C09148=1159.700,396.204,-85.224,-176.115,9.527,148.823
C09149=1159.704,395.957,-85.187,-176.115,9.525,148.822
C09150=1159.708,395.710,-85.150,-176.114,9.523,148.821
C09151=1159.712,395.462,-85.115,-176.114,9.520,148.821
C09152=1159.716,395.215,-85.078,-176.113,9.517,148.820
C09153=1159.720,394.968,-85.042,-176.112,9.515,148.819
C09154=1159.724,394.720,-85.005,-176.112,9.512,148.818
C09155=1159.728,394.473,-84.969,-176.112,9.510,148.818
C09156=1159.731,394.226,-84.932,-176.110,9.508,148.817
C09157=1159.736,393.979,-84.895,-176.110,9.505,148.816
C09158=1159.740,393.731,-84.859,-176.110,9.502,148.815
C09159=1159.743,393.484,-84.823,-176.109,9.500,148.814
C09160=1159.747,393.236,-84.786,-176.109,9.497,148.814
C09161=1159.750,392.989,-84.750,-176.108,9.495,148.813
C09162=1159.755,392.742,-84.713,-176.108,9.492,148.812
C09163=1159.759,392.495,-84.677,-176.107,9.489,148.811
C09164=1159.762,392.247,-84.641,-176.107,9.487,148.810
C09165=1159.766,392.000,-84.604,-176.107,9.484,148.809
C09166=1159.770,391.715,-84.562,-176.106,9.481,148.809
C09167=1159.775,391.429,-84.520,-176.106,9.477,148.808
C09168=1159.780,391.143,-84.479,-176.105,9.475,148.807
C09169=1159.784,390.858,-84.436,-176.106,9.471,148.806
C09170=1159.788,390.610,-84.400,-176.105,9.468,148.805
C09171=1159.792,390.363,-84.363,-176.105,9.465,148.804
C09172=1159.796,390.115,-84.326,-176.104,9.463,148.803
C09173=1159.799,389.867,-84.291,-176.104,9.460,148.803
C09174=1159.803,389.620,-84.254,-176.104,9.456,148.802
C09175=1159.807,389.373,-84.218,-176.104,9.454,148.801
C09176=1159.811,389.126,-84.181,-176.104,9.451,148.800
C09177=1159.814,388.879,-84.145,-176.104,9.448,148.799
C09178=1159.819,388.632,-84.108,-176.104,9.445,148.798
C09179=1159.822,388.384,-84.073,-176.104,9.441,148.798
C09180=1159.826,388.137,-84.036,-176.104,9.439,148.797
C09181=1159.831,387.889,-84.000,-176.104,9.435,148.796
C09182=1159.834,387.642,-83.964,-176.104,9.432,148.795
C09183=1159.838,387.395,-83.927,-176.104,9.429,148.794
C09184=1159.842,387.147,-83.891,-176.104,9.426,148.794
C09185=1159.846,386.900,-83.854,-176.104,9.423,148.793
C09186=1159.850,386.653,-83.819,-176.104,9.419,148.792
C09187=1159.854,386.406,-83.782,-176.105,9.416,148.791
C09188=1159.857,386.158,-83.746,-176.105,9.413,148.790
C09189=1159.861,385.911,-83.709,-176.105,9.410,148.790
C09190=1159.865,385.663,-83.674,-176.105,9.406,148.789
C09191=1159.869,385.416,-83.637,-176.106,9.403,148.788
C09192=1159.873,385.169,-83.601,-176.106,9.400,148.787
C09193=1159.877,384.921,-83.565,-176.106,9.396,148.786
C09194=1159.880,384.675,-83.528,-176.107,9.393,148.786
C09195=1159.885,384.427,-83.492,-176.107,9.389,148.785
C09196=1159.888,384.180,-83.456,-176.108,9.386,148.784
C09197=1159.892,383.932,-83.420,-176.109,9.382,148.783
C09198=1159.896,383.685,-83.384,-176.109,9.378,148.783
C09199=1159.900,383.437,-83.347,-176.110,9.375,148.782
C09200=1159.904,383.190,-83.312,-176.111,9.372,148.781
C09201=1159.908,382.943,-83.275,-176.112,9.368,148.780
C09202=1159.912,382.695,-83.239,-176.112,9.364,148.780
C09203=1159.916,382.448,-83.203,-176.112,9.361,148.779
C09204=1159.919,382.201,-83.167,-176.114,9.357,148.778
C09205=1159.923,381.954,-83.131,-176.114,9.354,148.777
C09206=1159.927,381.706,-83.095,-176.116,9.350,148.777
C09207=1159.931,381.458,-83.059,-176.116,9.346,148.776
C09208=1159.935,381.211,-83.022,-176.117,9.342,148.775
C09209=1159.939,380.964,-82.987,-176.118,9.339,148.775
C09210=1159.943,380.716,-82.950,-176.119,9.335,148.774
C09211=1159.947,380.470,-82.915,-176.120,9.332,148.773
C09212=1159.951,380.222,-82.879,-176.122,9.328,148.773
C09213=1159.955,379.975,-82.842,-176.123,9.324,148.772
C09214=1159.958,379.727,-82.807,-176.123,9.321,148.771
C09215=1159.963,379.480,-82.771,-176.125,9.317,148.771
C09216=1159.966,379.233,-82.734,-176.126,9.313,148.770
C09217=1159.970,378.985,-82.699,-176.127,9.309,148.769
C09218=1159.974,378.737,-82.663,-176.129,9.305,148.769
C09219=1159.978,378.490,-82.627,-176.130,9.302,148.768
C09220=1159.981,378.243,-82.591,-176.131,9.298,148.767
C09221=1159.986,377.995,-82.555,-176.133,9.294,148.767
C09222=1159.989,377.748,-82.519,-176.134,9.290,148.766
C09223=1159.994,377.501,-82.484,-176.135,9.286,148.765
C09224=1159.998,377.254,-82.447,-176.136,9.282,148.765
C09225=1160.001,377.006,-82.412,-176.138,9.278,148.764
C09226=1160.005,376.759,-82.376,-176.140,9.274,148.764
C09227=1160.009,376.511,-82.340,-176.141,9.270,148.763
C09228=1160.013,376.263,-82.304,-176.143,9.267,148.762
C09229=1160.016,376.017,-82.268,-176.144,9.263,148.762
C09230=1160.021,375.769,-82.232,-176.146,9.259,148.761
C09231=1160.025,375.522,-82.197,-176.147,9.255,148.761
C09232=1160.029,375.274,-82.161,-176.149,9.251,148.760
C09233=1160.032,375.027,-82.126,-176.150,9.247,148.759
C09234=1160.037,374.779,-82.089,-176.153,9.243,148.759
C09235=1160.040,374.532,-82.054,-176.154,9.239,148.758
C09236=1160.044,374.284,-82.018,-176.156,9.235,148.758
C09237=1160.048,374.037,-81.983,-176.158,9.232,148.757
C09238=1160.052,373.790,-81.948,-176.159,9.228,148.757
C09239=1160.056,373.542,-81.911,-176.161,9.223,148.756
C09240=1160.060,373.295,-81.876,-176.163,9.220,148.756
C09241=1160.064,373.047,-81.840,-176.165,9.216,148.755
C09242=1160.067,372.800,-81.805,-176.167,9.212,148.755
C09243=1160.072,372.553,-81.770,-176.169,9.208,148.754
C09244=1160.076,372.305,-81.734,-176.171,9.204,148.754
C09245=1160.080,372.057,-81.698,-176.172,9.200,148.753
C09246=1160.083,371.810,-81.662,-176.174,9.197,148.753
C09247=1160.087,371.562,-81.627,-176.177,9.192,148.752
C09248=1160.091,371.316,-81.592,-176.178,9.188,148.752
C09249=1160.095,371.068,-81.556,-176.180,9.185,148.751
C09250=1160.099,370.821,-81.521,-176.182,9.180,148.751
C09251=1160.102,370.573,-81.485,-176.184,9.177,148.750
C09252=1160.107,370.326,-81.449,-176.187,9.172,148.750
C09253=1160.111,370.079,-81.414,-176.189,9.169,148.750
C09254=1160.115,369.830,-81.379,-176.191,9.165,148.749
C09255=1160.119,369.583,-81.343,-176.193,9.161,148.749
C09256=1160.123,369.336,-81.308,-176.195,9.157,148.748
C09257=1160.126,369.089,-81.273,-176.197,9.153,148.748
C09258=1160.130,368.841,-81.237,-176.199,9.149,148.747
C09259=1160.134,368.593,-81.202,-176.202,9.145,148.747
C09260=1160.138,368.346,-81.167,-176.204,9.141,148.746
C09261=1160.142,368.099,-81.131,-176.206,9.138,148.746
C09262=1160.146,367.851,-81.096,-176.208,9.133,148.746
C09263=1160.150,367.604,-81.061,-176.210,9.130,148.745
C09264=1160.154,367.356,-81.026,-176.213,9.125,148.745
C09265=1160.158,367.109,-80.990,-176.215,9.122,148.744
C09266=1160.162,366.861,-80.956,-176.217,9.118,148.744
C09267=1160.166,366.614,-80.920,-176.219,9.114,148.744
C09268=1160.170,366.366,-80.885,-176.222,9.110,148.743
C09269=1160.173,366.118,-80.850,-176.224,9.106,148.743
C09270=1160.178,365.836,-80.810,-176.226,9.102,148.743
C09271=1160.183,365.553,-80.770,-176.229,9.097,148.742
C09272=1160.187,365.271,-80.730,-176.232,9.093,148.742
C09273=1160.192,364.988,-80.690,-176.235,9.088,148.741
C09274=1160.196,364.741,-80.654,-176.237,9.085,148.741
C09275=1160.200,364.493,-80.619,-176.240,9.081,148.741
C09276=1160.203,364.246,-80.585,-176.241,9.077,148.740
C09277=1160.207,363.998,-80.550,-176.244,9.073,148.740
C09278=1160.211,363.751,-80.515,-176.247,9.068,148.739
C09279=1160.215,363.503,-80.480,-176.249,9.065,148.739
C09280=1160.219,363.256,-80.444,-176.252,9.061,148.739
C09281=1160.224,363.008,-80.410,-176.254,9.057,148.738
C09282=1160.227,362.760,-80.375,-176.256,9.053,148.738
C09283=1160.231,362.513,-80.340,-176.259,9.050,148.738
C09284=1160.235,362.265,-80.305,-176.261,9.045,148.737
C09285=1160.239,362.018,-80.270,-176.263,9.042,148.737
C09286=1160.243,361.770,-80.235,-176.266,9.038,148.737
C09287=1160.247,361.523,-80.201,-176.268,9.034,148.736
C09288=1160.251,361.276,-80.166,-176.271,9.030,148.736
C09289=1160.255,361.028,-80.131,-176.273,9.027,148.736
C09290=1160.259,360.780,-80.096,-176.276,9.023,148.735
C09291=1160.263,360.533,-80.061,-176.278,9.019,148.735
C09292=1160.266,360.285,-80.027,-176.281,9.015,148.735
C09293=1160.271,360.038,-79.992,-176.283,9.012,148.735
C09294=1160.275,359.790,-79.957,-176.286,9.007,148.734
C09295=1160.278,359.543,-79.923,-176.288,9.004,148.734
C09296=1160.282,359.295,-79.888,-176.290,9.000,148.734
C09297=1160.287,359.047,-79.854,-176.293,8.996,148.733
C09298=1160.291,358.799,-79.819,-176.295,8.992,148.733
C09299=1160.294,358.553,-79.784,-176.298,8.989,148.733
C09300=1160.298,358.305,-79.749,-176.300,8.985,148.732
C09301=1160.303,358.057,-79.715,-176.302,8.981,148.732
C09302=1160.306,357.809,-79.681,-176.305,8.977,148.732
C09303=1160.311,357.562,-79.646,-176.307,8.974,148.731
C09304=1160.315,357.314,-79.611,-176.310,8.969,148.731
C09305=1160.319,357.067,-79.578,-176.312,8.966,148.731
C09306=1160.322,356.819,-79.543,-176.315,8.962,148.731
C09307=1160.326,356.572,-79.508,-176.317,8.959,148.730
C09308=1160.330,356.324,-79.473,-176.320,8.954,148.730
C09309=1160.335,356.077,-79.439,-176.322,8.951,148.730
C09310=1160.338,355.829,-79.405,-176.325,8.947,148.729
C09311=1160.342,355.581,-79.370,-176.327,8.943,148.729
C09312=1160.346,355.334,-79.336,-176.330,8.939,148.729
C09313=1160.350,355.086,-79.301,-176.332,8.936,148.728
C09314=1160.354,354.839,-79.268,-176.334,8.932,148.728
C09315=1160.358,354.591,-79.233,-176.337,8.928,148.728
C09316=1160.363,354.344,-79.198,-176.339,8.925,148.728
C09317=1160.366,354.095,-79.165,-176.342,8.921,148.727
C09318=1160.371,353.848,-79.130,-176.344,8.917,148.727
C09319=1160.374,353.600,-79.096,-176.347,8.913,148.727
C09320=1160.378,353.352,-79.062,-176.349,8.910,148.726
C09321=1160.382,353.105,-79.028,-176.351,8.906,148.726
C09322=1160.386,352.857,-78.993,-176.354,8.902,148.726
C09323=1160.390,352.610,-78.959,-176.357,8.899,148.726
C09324=1160.395,352.363,-78.925,-176.359,8.895,148.725
C09325=1160.398,352.114,-78.891,-176.361,8.891,148.725
C09326=1160.402,351.867,-78.857,-176.364,8.887,148.725
C09327=1160.406,351.619,-78.822,-176.366,8.884,148.725
C09328=1160.410,351.372,-78.788,-176.369,8.881,148.724
C09329=1160.415,351.124,-78.755,-176.371,8.876,148.724
C09330=1160.418,350.876,-78.721,-176.374,8.873,148.724
C09331=1160.422,350.629,-78.686,-176.376,8.869,148.723
C09332=1160.426,350.382,-78.652,-176.379,8.866,148.723
C09333=1160.430,350.133,-78.619,-176.381,8.862,148.723
C09334=1160.434,349.886,-78.584,-176.384,8.858,148.723
C09335=1160.438,349.639,-78.550,-176.386,8.855,148.722
C09336=1160.443,349.391,-78.517,-176.389,8.850,148.722
C09337=1160.446,349.143,-78.482,-176.391,8.847,148.722
C09338=1160.450,348.896,-78.448,-176.393,8.844,148.722
C09339=1160.455,348.648,-78.415,-176.396,8.840,148.721
C09340=1160.458,348.400,-78.380,-176.398,8.836,148.721
C09341=1160.462,348.152,-78.347,-176.401,8.832,148.721
C09342=1160.467,347.905,-78.313,-176.403,8.829,148.721
C09343=1160.471,347.657,-78.280,-176.406,8.825,148.720
C09344=1160.474,347.409,-78.245,-176.408,8.821,148.720
C09345=1160.478,347.162,-78.212,-176.411,8.818,148.720
C09346=1160.483,346.914,-78.178,-176.413,8.815,148.720
C09347=1160.487,346.667,-78.144,-176.416,8.811,148.719
C09348=1160.490,346.418,-78.110,-176.418,8.807,148.719
C09349=1160.495,346.170,-78.077,-176.421,8.803,148.719
C09350=1160.499,345.923,-78.043,-176.423,8.800,148.719
C09351=1160.503,345.676,-78.010,-176.426,8.797,148.718
C09352=1160.507,345.428,-77.975,-176.428,8.792,148.718
C09353=1160.511,345.180,-77.942,-176.430,8.789,148.718
C09354=1160.515,344.933,-77.908,-176.433,8.786,148.718
C09355=1160.519,344.685,-77.875,-176.436,8.782,148.717
C09356=1160.524,344.437,-77.841,-176.438,8.778,148.717
C09357=1160.527,344.189,-77.807,-176.440,8.775,148.717
C09358=1160.531,343.942,-77.774,-176.443,8.771,148.717
C09359=1160.536,343.694,-77.740,-176.445,8.768,148.716
C09360=1160.540,343.446,-77.706,-176.448,8.764,148.716
C09361=1160.544,343.199,-77.673,-176.451,8.760,148.716
C09362=1160.548,342.951,-77.640,-176.453,8.757,148.716
C09363=1160.551,342.703,-77.607,-176.456,8.753,148.716
C09364=1160.555,342.455,-77.573,-176.458,8.750,148.715
C09365=1160.560,342.207,-77.539,-176.460,8.746,148.715
C09366=1160.564,341.960,-77.506,-176.463,8.742,148.715
C09367=1160.568,341.712,-77.473,-176.466,8.739,148.715
C09368=1160.572,341.465,-77.439,-176.468,8.736,148.714
C09369=1160.576,341.217,-77.406,-176.471,8.732,148.714
C09370=1160.580,340.969,-77.372,-176.473,8.728,148.714
C09371=1160.584,340.721,-77.339,-176.475,8.725,148.714
C09372=1160.588,340.473,-77.306,-176.478,8.721,148.714
C09373=1160.592,340.226,-77.273,-176.481,8.718,148.713
C09374=1160.597,339.946,-77.235,-176.483,8.713,148.713
C09375=1160.602,339.666,-77.198,-176.486,8.709,148.713
C09376=1160.606,339.387,-77.160,-176.489,8.705,148.713
C09377=1160.611,339.107,-77.123,-176.491,8.702,148.712
C09378=1160.615,338.859,-77.089,-176.494,8.698,148.712
C09379=1160.618,338.611,-77.056,-176.497,8.695,148.712
C09380=1160.623,338.363,-77.023,-176.499,8.691,148.712
C09381=1160.627,338.116,-76.990,-176.502,8.687,148.711
C09382=1160.631,337.868,-76.956,-176.504,8.684,148.711
C09383=1160.635,337.620,-76.923,-176.506,8.681,148.711
C09384=1160.639,337.372,-76.890,-176.509,8.676,148.711
C09385=1160.643,337.125,-76.857,-176.512,8.673,148.711
C09386=1160.647,336.877,-76.824,-176.514,8.670,148.710
C09387=1160.651,336.629,-76.791,-176.517,8.666,148.710
C09388=1160.656,336.381,-76.757,-176.519,8.663,148.710
C09389=1160.660,336.134,-76.724,-176.521,8.659,148.710
C09390=1160.664,335.886,-76.691,-176.524,8.656,148.710
C09391=1160.668,335.638,-76.659,-176.527,8.652,148.709
C09392=1160.672,335.390,-76.626,-176.529,8.649,148.709
C09393=1160.676,335.142,-76.593,-176.532,8.646,148.709
C09394=1160.680,334.895,-76.560,-176.535,8.641,148.709
C09395=1160.684,334.647,-76.527,-176.537,8.638,148.709
C09396=1160.688,334.399,-76.494,-176.539,8.635,148.708
C09397=1160.693,334.151,-76.461,-176.541,8.632,148.708
C09398=1160.696,333.904,-76.429,-176.544,8.628,148.708
C09399=1160.700,333.656,-76.395,-176.547,8.624,148.708
C09400=1160.704,333.408,-76.362,-176.549,8.621,148.708
C09401=1160.709,333.160,-76.330,-176.552,8.617,148.708
C09402=1160.713,332.912,-76.297,-176.555,8.614,148.707
C09403=1160.716,332.665,-76.264,-176.557,8.611,148.707
C09404=1160.721,332.416,-76.232,-176.559,8.607,148.707
C09405=1160.725,332.168,-76.198,-176.562,8.603,148.707
C09406=1160.729,331.921,-76.165,-176.564,8.600,148.706
C09407=1160.733,331.673,-76.133,-176.567,8.597,148.706
C09408=1160.738,331.426,-76.101,-176.569,8.593,148.706
C09409=1160.742,331.178,-76.068,-176.572,8.590,148.706
C09410=1160.745,330.930,-76.036,-176.575,8.586,148.706
C09411=1160.750,330.682,-76.003,-176.577,8.583,148.706
C09412=1160.754,330.434,-75.970,-176.580,8.579,148.705
C09413=1160.758,330.186,-75.937,-176.582,8.576,148.705
C09414=1160.762,329.939,-75.904,-176.584,8.572,148.705
C09415=1160.766,329.690,-75.872,-176.587,8.569,148.705
C09416=1160.770,329.443,-75.839,-176.590,8.565,148.705
C09417=1160.774,329.195,-75.807,-176.592,8.562,148.705
C09418=1160.779,328.948,-75.774,-176.595,8.559,148.704
C09419=1160.782,328.700,-75.742,-176.597,8.555,148.704
C09420=1160.786,328.452,-75.709,-176.600,8.551,148.704
C09421=1160.791,328.203,-75.677,-176.602,8.548,148.704
C09422=1160.795,327.955,-75.645,-176.605,8.545,148.704
C09423=1160.799,327.708,-75.612,-176.607,8.542,148.704
C09424=1160.804,327.460,-75.580,-176.610,8.538,148.703
C09425=1160.807,327.213,-75.547,-176.612,8.534,148.703
C09426=1160.812,326.964,-75.515,-176.615,8.531,148.703
C09427=1160.815,326.716,-75.483,-176.617,8.528,148.703
C09428=1160.819,326.468,-75.450,-176.620,8.524,148.703
C09429=1160.823,326.220,-75.418,-176.622,8.521,148.702
C09430=1160.828,325.973,-75.386,-176.625,8.517,148.702
C09431=1160.832,325.725,-75.353,-176.628,8.514,148.702
C09432=1160.836,325.477,-75.321,-176.630,8.511,148.702
C09433=1160.840,325.229,-75.289,-176.633,8.507,148.702
C09434=1160.844,324.981,-75.256,-176.635,8.504,148.702
C09435=1160.848,324.734,-75.224,-176.638,8.501,148.702
C09436=1160.853,324.486,-75.192,-176.640,8.497,148.701
C09437=1160.856,324.238,-75.160,-176.643,8.493,148.701
C09438=1160.861,323.989,-75.127,-176.645,8.490,148.701
C09439=1160.865,323.742,-75.095,-176.648,8.487,148.701
C09440=1160.869,323.494,-75.063,-176.650,8.484,148.701
C09441=1160.873,323.246,-75.031,-176.653,8.480,148.701
C09442=1160.877,322.998,-74.999,-176.655,8.476,148.700
C09443=1160.881,322.750,-74.967,-176.658,8.473,148.700
C09444=1160.885,322.502,-74.935,-176.661,8.470,148.700
C09445=1160.890,322.255,-74.902,-176.663,8.467,148.700
C09446=1160.893,322.007,-74.870,-176.666,8.463,148.700
C09447=1160.898,321.759,-74.839,-176.668,8.460,148.700
C09448=1160.902,321.511,-74.806,-176.671,8.457,148.700
C09449=1160.906,321.263,-74.774,-176.673,8.453,148.699
C09450=1160.909,321.015,-74.743,-176.676,8.450,148.699
C09451=1160.914,320.767,-74.711,-176.679,8.446,148.699
C09452=1160.918,320.519,-74.679,-176.681,8.443,148.699
C09453=1160.922,320.271,-74.647,-176.684,8.440,148.699
C09454=1160.927,320.023,-74.615,-176.686,8.437,148.699
C09455=1160.931,319.775,-74.583,-176.688,8.433,148.699
C09456=1160.934,319.527,-74.551,-176.691,8.429,148.698
C09457=1160.939,319.280,-74.519,-176.694,8.426,148.698
C09458=1160.943,319.032,-74.487,-176.696,8.423,148.698
C09459=1160.947,318.784,-74.455,-176.699,8.420,148.698
C09460=1160.952,318.536,-74.423,-176.701,8.417,148.698
C09461=1160.956,318.287,-74.392,-176.704,8.413,148.698
C09462=1160.960,318.039,-74.360,-176.706,8.409,148.698
C09463=1160.964,317.792,-74.329,-176.709,8.406,148.698
C09464=1160.968,317.544,-74.297,-176.712,8.403,148.697
C09465=1160.972,317.296,-74.265,-176.714,8.400,148.697
C09466=1160.976,317.048,-74.233,-176.717,8.397,148.697
C09467=1160.980,316.800,-74.201,-176.719,8.393,148.697
C09468=1160.985,316.552,-74.170,-176.722,8.389,148.697
C09469=1160.989,316.304,-74.138,-176.725,8.386,148.697
C09470=1160.993,316.056,-74.106,-176.727,8.383,148.697
C09471=1160.997,315.809,-74.075,-176.729,8.380,148.696
C09472=1161.001,315.560,-74.044,-176.732,8.377,148.696
C09473=1161.005,315.313,-74.012,-176.735,8.373,148.696
C09474=1161.009,315.064,-73.980,-176.737,8.370,148.696
C09475=1161.013,314.817,-73.949,-176.740,8.367,148.696
C09476=1161.018,314.568,-73.917,-176.742,8.363,148.696
C09477=1161.022,314.320,-73.885,-176.745,8.360,148.696
C09478=1161.027,314.043,-73.850,-176.748,8.356,148.696
C09479=1161.032,313.766,-73.815,-176.751,8.352,148.695
C09480=1161.036,313.489,-73.780,-176.753,8.349,148.695
C09481=1161.040,313.212,-73.745,-176.756,8.345,148.695
C09482=1161.044,312.964,-73.713,-176.759,8.342,148.695
C09483=1161.049,312.716,-73.683,-176.761,8.339,148.695
C09484=1161.053,312.467,-73.650,-176.764,8.336,148.695
C09485=1161.058,312.220,-73.619,-176.767,8.332,148.695
C09486=1161.062,311.971,-73.587,-176.769,8.328,148.695
C09487=1161.066,311.724,-73.557,-176.772,8.325,148.695
C09488=1161.070,311.475,-73.525,-176.774,8.322,148.694
C09489=1161.075,311.228,-73.494,-176.777,8.319,148.694
C09490=1161.078,310.979,-73.462,-176.779,8.316,148.694
C09491=1161.083,310.732,-73.432,-176.782,8.313,148.694
C09492=1161.087,310.483,-73.400,-176.785,8.309,148.694
C09493=1161.091,310.236,-73.369,-176.787,8.306,148.694
C09494=1161.095,309.988,-73.337,-176.790,8.303,148.694
C09495=1161.099,309.740,-73.306,-176.792,8.299,148.694
C09496=1161.103,309.491,-73.275,-176.795,8.296,148.694
C09497=1161.108,309.244,-73.244,-176.797,8.293,148.694
C09498=1161.111,308.995,-73.213,-176.800,8.290,148.693
C09499=1161.115,308.748,-73.182,-176.803,8.286,148.693
C09500=1161.120,308.500,-73.151,-176.805,8.283,148.693
C09501=1161.124,308.251,-73.120,-176.808,8.280,148.693
C09502=1161.128,308.004,-73.088,-176.810,8.276,148.693
C09503=1161.132,307.755,-73.057,-176.813,8.274,148.693
C09504=1161.137,307.507,-73.026,-176.815,8.270,148.693
C09505=1161.142,307.259,-72.996,-176.818,8.267,148.693
C09506=1161.145,307.011,-72.964,-176.820,8.264,148.693
C09507=1161.150,306.763,-72.933,-176.824,8.260,148.693
C09508=1161.153,306.515,-72.902,-176.826,8.257,148.692
C09509=1161.158,306.267,-72.872,-176.829,8.254,148.692
C09510=1161.162,306.020,-72.840,-176.831,8.251,148.692
C09511=1161.166,305.771,-72.809,-176.833,8.247,148.692
C09512=1161.171,305.523,-72.778,-176.836,8.244,148.692
C09513=1161.175,305.275,-72.748,-176.838,8.241,148.692
C09514=1161.179,305.027,-72.717,-176.841,8.238,148.692
C09515=1161.183,304.779,-72.686,-176.843,8.235,148.692
C09516=1161.187,304.531,-72.654,-176.847,8.231,148.692
C09517=1161.192,304.283,-72.624,-176.849,8.228,148.692
C09518=1161.196,304.035,-72.593,-176.852,8.225,148.692
C09519=1161.199,303.787,-72.562,-176.854,8.222,148.691
C09520=1161.204,303.539,-72.532,-176.857,8.219,148.691
C09521=1161.209,303.291,-72.501,-176.859,8.215,148.691
C09522=1161.213,303.043,-72.470,-176.862,8.212,148.691
C09523=1161.217,302.794,-72.440,-176.865,8.209,148.691
C09524=1161.221,302.546,-72.409,-176.867,8.206,148.691
C09525=1161.226,302.298,-72.378,-176.870,8.203,148.691
C09526=1161.229,302.050,-72.347,-176.873,8.199,148.691
C09527=1161.234,301.802,-72.317,-176.875,8.196,148.691
C09528=1161.238,301.554,-72.286,-176.878,8.193,148.691
C09529=1161.242,301.306,-72.256,-176.880,8.190,148.691
C09530=1161.246,301.058,-72.225,-176.883,8.187,148.691
C09531=1161.251,300.810,-72.194,-176.886,8.184,148.691
C09532=1161.255,300.562,-72.164,-176.888,8.180,148.691
C09533=1161.259,300.314,-72.133,-176.891,8.177,148.691
C09534=1161.264,300.065,-72.103,-176.893,8.174,148.690
C09535=1161.267,299.817,-72.072,-176.896,8.171,148.690
C09536=1161.272,299.569,-72.042,-176.898,8.168,148.690
C09537=1161.276,299.321,-72.010,-176.901,8.164,148.690
C09538=1161.280,299.073,-71.980,-176.904,8.161,148.690
C09539=1161.285,298.825,-71.950,-176.906,8.158,148.690
C09540=1161.289,298.577,-71.920,-176.909,8.155,148.690
C09541=1161.293,298.329,-71.889,-176.911,8.151,148.690
C09542=1161.297,298.081,-71.859,-176.914,8.149,148.690
C09543=1161.301,297.833,-71.828,-176.916,8.145,148.690
C09544=1161.305,297.585,-71.798,-176.919,8.142,148.690
C09545=1161.310,297.336,-71.768,-176.922,8.139,148.690
C09546=1161.315,297.088,-71.737,-176.924,8.136,148.690
C09547=1161.318,296.840,-71.707,-176.927,8.133,148.690
C09548=1161.323,296.591,-71.676,-176.929,8.130,148.689
C09549=1161.327,296.344,-71.646,-176.932,8.127,148.690
C09550=1161.331,296.096,-71.616,-176.935,8.124,148.690
C09551=1161.335,295.848,-71.586,-176.937,8.121,148.689
C09552=1161.339,295.600,-71.556,-176.940,8.117,148.689
C09553=1161.343,295.351,-71.525,-176.943,8.113,148.689
C09554=1161.348,295.103,-71.495,-176.945,8.111,148.689
C09555=1161.352,294.855,-71.465,-176.948,8.108,148.689
C09556=1161.356,294.607,-71.435,-176.950,8.104,148.689
C09557=1161.361,294.359,-71.404,-176.953,8.101,148.689
C09558=1161.365,294.111,-71.374,-176.956,8.098,148.689
C09559=1161.369,293.863,-71.345,-176.958,8.095,148.689
C09560=1161.373,293.614,-71.314,-176.961,8.092,148.689
C09561=1161.377,293.366,-71.284,-176.963,8.089,148.689
C09562=1161.382,293.118,-71.253,-176.966,8.086,148.689
C09563=1161.386,292.870,-71.224,-176.969,8.083,148.689
C09564=1161.390,292.622,-71.194,-176.971,8.080,148.689
C09565=1161.395,292.374,-71.164,-176.974,8.077,148.689
C09566=1161.399,292.126,-71.134,-176.977,8.074,148.689
C09567=1161.403,291.878,-71.104,-176.979,8.070,148.689
C09568=1161.408,291.629,-71.074,-176.982,8.067,148.689
C09569=1161.412,291.381,-71.044,-176.984,8.064,148.689
C09570=1161.415,291.132,-71.014,-176.987,8.061,148.688
C09571=1161.419,290.885,-70.984,-176.990,8.058,148.689
C09572=1161.424,290.636,-70.954,-176.992,8.055,148.689
C09573=1161.428,290.388,-70.924,-176.995,8.052,148.688
C09574=1161.432,290.140,-70.894,-176.997,8.049,148.688
C09575=1161.437,289.892,-70.864,-177.001,8.045,148.688
C09576=1161.441,289.643,-70.835,-177.003,8.042,148.688
C09577=1161.445,289.396,-70.805,-177.006,8.039,148.688
C09578=1161.449,289.148,-70.775,-177.008,8.036,148.688
C09579=1161.454,288.899,-70.745,-177.011,8.033,148.688
C09580=1161.458,288.651,-70.716,-177.014,8.030,148.688
C09581=1161.462,288.403,-70.685,-177.016,8.027,148.688
C09582=1161.467,288.128,-70.653,-177.019,8.024,148.688
C09583=1161.472,287.853,-70.620,-177.022,8.020,148.688
C09584=1161.477,287.577,-70.587,-177.025,8.017,148.688
C09585=1161.481,287.303,-70.554,-177.027,8.014,148.688
C09586=1161.486,287.054,-70.524,-177.030,8.011,148.688
C09587=1161.490,286.806,-70.495,-177.032,8.008,148.688
C09588=1161.494,286.558,-70.465,-177.035,8.005,148.688
C09589=1161.498,286.310,-70.436,-177.038,8.002,148.688
C09590=1161.502,286.061,-70.406,-177.040,7.998,148.688
C09591=1161.507,285.813,-70.376,-177.043,7.995,148.688
C09592=1161.511,285.565,-70.346,-177.046,7.993,148.688
C09593=1161.515,285.317,-70.317,-177.048,7.989,148.688
C09594=1161.520,285.069,-70.288,-177.051,7.986,148.688
C09595=1161.524,284.821,-70.258,-177.054,7.983,148.688
C09596=1161.528,284.573,-70.229,-177.056,7.980,148.688
C09597=1161.533,284.325,-70.199,-177.059,7.977,148.688
C09598=1161.537,284.076,-70.170,-177.061,7.974,148.688
C09599=1161.541,283.828,-70.140,-177.064,7.971,148.688
C09600=1161.545,283.580,-70.111,-177.067,7.968,148.688
C09601=1161.549,283.331,-70.081,-177.069,7.965,148.688
C09602=1161.554,283.083,-70.052,-177.072,7.962,148.688
C09603=1161.558,282.835,-70.022,-177.075,7.959,148.688
C09604=1161.563,282.586,-69.992,-177.078,7.956,148.688
C09605=1161.568,282.338,-69.964,-177.080,7.953,148.688
C09606=1161.572,282.090,-69.935,-177.083,7.950,148.688
C09607=1161.576,281.842,-69.905,-177.085,7.947,148.688
C09608=1161.580,281.593,-69.876,-177.088,7.944,148.688
C09609=1161.584,281.345,-69.847,-177.090,7.941,148.688
C09610=1161.588,281.097,-69.817,-177.093,7.938,148.688
C09611=1161.592,280.849,-69.788,-177.096,7.935,148.688
C09612=1161.597,280.601,-69.760,-177.099,7.932,148.688
C09613=1161.601,280.352,-69.730,-177.101,7.928,148.688
C09614=1161.605,280.104,-69.701,-177.104,7.925,148.688
C09615=1161.610,279.856,-69.671,-177.106,7.922,148.688
C09616=1161.614,279.608,-69.642,-177.109,7.920,148.688
C09617=1161.619,279.359,-69.613,-177.112,7.917,148.688
C09618=1161.623,279.111,-69.584,-177.114,7.913,148.688
C09619=1161.627,278.863,-69.554,-177.117,7.910,148.688
C09620=1161.631,278.615,-69.525,-177.120,7.907,148.688
C09621=1161.635,278.366,-69.497,-177.123,7.904,148.688
C09622=1161.639,278.118,-69.467,-177.125,7.901,148.688
C09623=1161.644,277.870,-69.438,-177.128,7.898,148.688
C09624=1161.649,277.621,-69.410,-177.130,7.895,148.688
C09625=1161.653,277.373,-69.380,-177.133,7.892,148.688
C09626=1161.657,277.125,-69.351,-177.136,7.889,148.688
C09627=1161.661,276.877,-69.323,-177.139,7.886,148.688
C09628=1161.666,276.629,-69.293,-177.141,7.883,148.688
C09629=1161.670,276.380,-69.265,-177.144,7.880,148.688
C09630=1161.674,276.131,-69.235,-177.146,7.877,148.688
C09631=1161.679,275.884,-69.206,-177.149,7.875,148.688
C09632=1161.683,275.635,-69.178,-177.151,7.872,148.688
C09633=1161.687,275.387,-69.149,-177.154,7.869,148.688
C09634=1161.691,275.138,-69.120,-177.156,7.866,148.688
C09635=1161.696,274.891,-69.091,-177.159,7.863,148.688
C09636=1161.700,274.642,-69.063,-177.162,7.860,148.688
C09637=1161.704,274.394,-69.033,-177.165,7.857,148.688
C09638=1161.709,274.146,-69.005,-177.168,7.854,148.688
C09639=1161.713,273.898,-68.976,-177.170,7.851,148.688
C09640=1161.717,273.649,-68.947,-177.173,7.848,148.688
C09641=1161.722,273.400,-68.918,-177.175,7.845,148.688
C09642=1161.726,273.153,-68.890,-177.178,7.842,148.688
C09643=1161.730,272.904,-68.861,-177.181,7.839,148.688
C09644=1161.734,272.655,-68.832,-177.184,7.836,148.688
C09645=1161.739,272.408,-68.804,-177.186,7.833,148.688
C09646=1161.743,272.159,-68.775,-177.189,7.830,148.688
C09647=1161.747,271.910,-68.746,-177.191,7.828,148.688
C09648=1161.752,271.663,-68.718,-177.194,7.825,148.688
C09649=1161.756,271.414,-68.689,-177.196,7.822,148.688
C09650=1161.760,271.165,-68.660,-177.199,7.819,148.688
C09651=1161.765,270.918,-68.632,-177.202,7.816,148.688
C09652=1161.769,270.669,-68.603,-177.205,7.813,148.688
C09653=1161.773,270.421,-68.575,-177.207,7.810,148.688
C09654=1161.778,270.172,-68.546,-177.210,7.807,148.688
C09655=1161.782,269.924,-68.517,-177.213,7.804,148.688
C09656=1161.787,269.676,-68.490,-177.216,7.801,148.688
C09657=1161.791,269.427,-68.460,-177.218,7.798,148.688
C09658=1161.795,269.180,-68.432,-177.220,7.796,148.688
C09659=1161.800,268.931,-68.404,-177.223,7.793,148.688
C09660=1161.803,268.682,-68.375,-177.226,7.790,148.688
C09661=1161.808,268.434,-68.347,-177.228,7.787,148.688
C09662=1161.812,268.185,-68.319,-177.231,7.784,148.689
C09663=1161.817,267.938,-68.290,-177.234,7.781,148.689
C09664=1161.821,267.689,-68.262,-177.237,7.778,148.689
C09665=1161.826,267.441,-68.233,-177.239,7.775,148.689
C09666=1161.830,267.192,-68.205,-177.242,7.772,148.689
C09667=1161.834,266.944,-68.176,-177.245,7.769,148.689
C09668=1161.838,266.696,-68.149,-177.247,7.767,148.689
C09669=1161.843,266.447,-68.120,-177.250,7.764,148.689
C09670=1161.847,266.199,-68.092,-177.253,7.761,148.689
C09671=1161.852,265.950,-68.063,-177.255,7.758,148.689
C09672=1161.856,265.702,-68.036,-177.258,7.755,148.689
C09673=1161.861,265.453,-68.007,-177.261,7.752,148.689
C09674=1161.865,265.205,-67.979,-177.263,7.749,148.689
C09675=1161.869,264.957,-67.951,-177.266,7.746,148.689
C09676=1161.874,264.709,-67.923,-177.269,7.743,148.689
C09677=1161.878,264.460,-67.894,-177.271,7.741,148.689
C09678=1161.883,264.212,-67.866,-177.274,7.738,148.689
C09679=1161.886,263.963,-67.838,-177.277,7.735,148.689
C09680=1161.891,263.715,-67.810,-177.279,7.732,148.689
C09681=1161.895,263.467,-67.781,-177.282,7.729,148.689
C09682=1161.900,263.219,-67.754,-177.285,7.726,148.689
C09683=1161.903,262.970,-67.726,-177.288,7.723,148.690
C09684=1161.909,262.721,-67.698,-177.290,7.720,148.690
C09685=1161.913,262.473,-67.670,-177.293,7.718,148.690
C09686=1161.918,262.200,-67.639,-177.296,7.714,148.690
C09687=1161.922,261.927,-67.608,-177.299,7.711,148.690
C09688=1161.927,261.654,-67.577,-177.301,7.708,148.690
C09689=1161.931,261.381,-67.547,-177.304,7.705,148.690
C09690=1161.937,261.133,-67.518,-177.307,7.702,148.690
C09691=1161.941,260.883,-67.491,-177.310,7.699,148.690
C09692=1161.945,260.635,-67.463,-177.312,7.696,148.690
C09693=1161.949,260.387,-67.435,-177.315,7.693,148.690
C09694=1161.954,260.138,-67.407,-177.318,7.691,148.690
C09695=1161.958,259.890,-67.380,-177.321,7.688,148.690
C09696=1161.962,259.642,-67.351,-177.323,7.685,148.690
C09697=1161.967,259.394,-67.324,-177.326,7.683,148.690
C09698=1161.971,259.144,-67.296,-177.328,7.680,148.690
C09699=1161.976,258.896,-67.268,-177.332,7.677,148.691
C09700=1161.980,258.648,-67.240,-177.334,7.674,148.691
C09701=1161.984,258.399,-67.213,-177.337,7.671,148.691
C09702=1161.988,258.151,-67.185,-177.339,7.669,148.691
C09703=1161.992,257.902,-67.157,-177.342,7.666,148.691
C09704=1161.998,257.654,-67.129,-177.345,7.663,148.691
C09705=1162.002,257.406,-67.101,-177.348,7.660,148.691
C09706=1162.006,257.157,-67.074,-177.350,7.657,148.691
C09707=1162.010,256.909,-67.046,-177.353,7.654,148.691
C09708=1162.015,256.661,-67.019,-177.355,7.652,148.691
C09709=1162.019,256.412,-66.991,-177.358,7.649,148.691
C09710=1162.023,256.163,-66.964,-177.361,7.646,148.691
C09711=1162.028,255.916,-66.936,-177.364,7.643,148.692
C09712=1162.032,255.667,-66.909,-177.366,7.640,148.692
C09713=1162.037,255.418,-66.880,-177.369,7.637,148.692
C09714=1162.042,255.170,-66.853,-177.371,7.635,148.692
C09715=1162.046,254.922,-66.825,-177.374,7.632,148.692
C09716=1162.050,254.673,-66.798,-177.377,7.629,148.692
C09717=1162.054,254.425,-66.770,-177.380,7.626,148.692
C09718=1162.059,254.176,-66.743,-177.382,7.623,148.692
C09719=1162.063,253.927,-66.716,-177.385,7.622,148.692
C09720=1162.067,253.679,-66.688,-177.388,7.619,148.692
C09721=1162.072,253.431,-66.661,-177.391,7.616,148.692
C09722=1162.077,253.182,-66.634,-177.393,7.613,148.692
C09723=1162.080,252.934,-66.606,-177.396,7.610,148.693
C09724=1162.085,252.685,-66.579,-177.398,7.608,148.693
C09725=1162.090,252.437,-66.552,-177.401,7.605,148.693
C09726=1162.094,252.189,-66.524,-177.404,7.602,148.693
C09727=1162.098,251.940,-66.496,-177.407,7.599,148.693
C09728=1162.103,251.691,-66.469,-177.409,7.596,148.693
C09729=1162.107,251.443,-66.441,-177.412,7.594,148.693
C09730=1162.111,251.195,-66.415,-177.415,7.591,148.693
C09731=1162.116,250.947,-66.388,-177.418,7.588,148.693
C09732=1162.120,250.697,-66.361,-177.420,7.585,148.693
C09733=1162.124,250.449,-66.333,-177.423,7.582,148.693
C09734=1162.129,250.201,-66.306,-177.425,7.580,148.694
C09735=1162.133,249.952,-66.279,-177.428,7.577,148.694
C09736=1162.138,249.704,-66.252,-177.431,7.574,148.694
C09737=1162.142,249.455,-66.224,-177.434,7.571,148.694
C09738=1162.147,249.206,-66.197,-177.437,7.569,148.694
C09739=1162.150,248.959,-66.170,-177.439,7.566,148.694
C09740=1162.155,248.710,-66.143,-177.442,7.564,148.694
C09741=1162.160,248.462,-66.116,-177.445,7.561,148.694
C09742=1162.164,248.213,-66.089,-177.447,7.558,148.694
C09743=1162.168,247.964,-66.061,-177.449,7.556,148.694
C09744=1162.173,247.716,-66.034,-177.452,7.553,148.695
C09745=1162.177,247.467,-66.008,-177.455,7.550,148.695
C09746=1162.182,247.219,-65.981,-177.458,7.547,148.695
C09747=1162.186,246.970,-65.954,-177.460,7.545,148.695
C09748=1162.191,246.722,-65.927,-177.463,7.542,148.695
C09749=1162.196,246.473,-65.899,-177.466,7.539,148.695
C09750=1162.199,246.224,-65.873,-177.469,7.536,148.695
C09751=1162.204,245.976,-65.846,-177.471,7.533,148.695
C09752=1162.208,245.727,-65.819,-177.474,7.531,148.696
C09753=1162.212,245.479,-65.792,-177.477,7.528,148.696
C09754=1162.217,245.231,-65.765,-177.480,7.525,148.696
C09755=1162.222,244.982,-65.738,-177.482,7.522,148.696
C09756=1162.226,244.734,-65.711,-177.485,7.520,148.696
C09757=1162.230,244.486,-65.684,-177.488,7.518,148.696
C09758=1162.235,244.237,-65.657,-177.491,7.515,148.696
C09759=1162.239,243.989,-65.630,-177.493,7.512,148.696
C09760=1162.244,243.740,-65.605,-177.496,7.510,148.696
C09761=1162.248,243.491,-65.577,-177.498,7.507,148.696
C09762=1162.253,243.243,-65.550,-177.501,7.504,148.697
C09763=1162.256,242.994,-65.524,-177.504,7.502,148.697
C09764=1162.261,242.745,-65.497,-177.507,7.499,148.697
C09765=1162.266,242.497,-65.469,-177.509,7.496,148.697
C09766=1162.270,242.248,-65.444,-177.512,7.493,148.697
C09767=1162.274,242.000,-65.417,-177.514,7.491,148.697
C09768=1162.278,241.751,-65.390,-177.518,7.488,148.697
C09769=1162.283,241.503,-65.363,-177.520,7.485,148.698
C09770=1162.288,241.254,-65.337,-177.523,7.483,148.698
C09771=1162.292,241.006,-65.310,-177.525,7.480,148.698
C09772=1162.297,240.757,-65.283,-177.528,7.478,148.698
C09773=1162.301,240.508,-65.258,-177.531,7.475,148.698
C09774=1162.305,240.260,-65.230,-177.533,7.473,148.698
C09775=1162.309,240.012,-65.204,-177.536,7.470,148.698
C09776=1162.314,239.763,-65.178,-177.539,7.467,148.698
C09777=1162.319,239.514,-65.151,-177.542,7.464,148.699
C09778=1162.323,239.266,-65.124,-177.544,7.462,148.699
C09779=1162.328,239.017,-65.098,-177.547,7.459,148.699
C09780=1162.332,238.769,-65.071,-177.550,7.456,148.699
C09781=1162.337,238.521,-65.045,-177.553,7.454,148.699
C09782=1162.341,238.272,-65.019,-177.555,7.451,148.699
C09783=1162.346,238.024,-64.992,-177.558,7.449,148.699
C09784=1162.350,237.775,-64.966,-177.561,7.446,148.699
C09785=1162.355,237.526,-64.939,-177.564,7.444,148.700
C09786=1162.359,237.277,-64.913,-177.566,7.441,148.700
C09787=1162.363,237.029,-64.887,-177.569,7.438,148.700
C09788=1162.368,236.780,-64.860,-177.571,7.436,148.700
C09789=1162.372,236.532,-64.834,-177.575,7.433,148.700
C09790=1162.377,236.260,-64.805,-177.577,7.430,148.700
C09791=1162.382,235.988,-64.777,-177.581,7.428,148.701
C09792=1162.387,235.717,-64.747,-177.583,7.425,148.701
C09793=1162.391,235.445,-64.719,-177.586,7.422,148.701
C09794=1162.396,235.196,-64.692,-177.589,7.419,148.701
C09795=1162.400,234.948,-64.666,-177.592,7.416,148.701
C09796=1162.405,234.699,-64.641,-177.594,7.414,148.701
C09797=1162.410,234.451,-64.614,-177.597,7.411,148.701
C09798=1162.414,234.202,-64.588,-177.600,7.409,148.702
C09799=1162.418,233.954,-64.562,-177.602,7.406,148.702
C09800=1162.423,233.705,-64.535,-177.605,7.403,148.702
C09801=1162.427,233.456,-64.510,-177.608,7.401,148.702
C09802=1162.431,233.208,-64.483,-177.611,7.399,148.702
C09803=1162.436,232.959,-64.457,-177.613,7.396,148.702
C09804=1162.441,232.711,-64.431,-177.617,7.393,148.703
C09805=1162.445,232.462,-64.406,-177.619,7.391,148.703
C09806=1162.449,232.214,-64.379,-177.622,7.388,148.703
C09807=1162.454,231.965,-64.353,-177.624,7.385,148.703
C09808=1162.458,231.716,-64.327,-177.627,7.383,148.703
C09809=1162.463,231.468,-64.302,-177.630,7.380,148.703
C09810=1162.468,231.219,-64.275,-177.632,7.378,148.703
C09811=1162.472,230.970,-64.249,-177.635,7.376,148.704
C09812=1162.476,230.722,-64.223,-177.638,7.373,148.704
C09813=1162.480,230.473,-64.197,-177.640,7.371,148.704
C09814=1162.485,230.225,-64.172,-177.643,7.368,148.704
C09815=1162.490,229.976,-64.145,-177.646,7.365,148.704
C09816=1162.494,229.727,-64.119,-177.648,7.363,148.704
C09817=1162.498,229.479,-64.093,-177.652,7.360,148.705
C09818=1162.503,229.231,-64.068,-177.654,7.357,148.705
C09819=1162.507,228.982,-64.042,-177.657,7.355,148.705
C09820=1162.512,228.733,-64.016,-177.660,7.353,148.705
C09821=1162.517,228.484,-63.990,-177.663,7.350,148.705
C09822=1162.521,228.236,-63.965,-177.665,7.348,148.705
C09823=1162.526,227.987,-63.939,-177.668,7.345,148.706
C09824=1162.530,227.738,-63.913,-177.670,7.343,148.706
C09825=1162.534,227.489,-63.888,-177.673,7.340,148.706
C09826=1162.539,227.241,-63.862,-177.676,7.337,148.706
C09827=1162.544,226.992,-63.836,-177.678,7.335,148.706
C09828=1162.548,226.743,-63.810,-177.682,7.333,148.707
C09829=1162.553,226.495,-63.785,-177.684,7.331,148.707
C09830=1162.557,226.246,-63.759,-177.687,7.328,148.707
C09831=1162.561,225.998,-63.733,-177.690,7.325,148.707
C09832=1162.566,225.749,-63.707,-177.692,7.323,148.707
C09833=1162.570,225.501,-63.682,-177.695,7.320,148.707
C09834=1162.575,225.252,-63.656,-177.698,7.317,148.708
C09835=1162.579,225.003,-63.631,-177.700,7.315,148.708
C09836=1162.584,224.755,-63.605,-177.704,7.313,148.708
C09837=1162.588,224.506,-63.579,-177.706,7.310,148.708
C09838=1162.592,224.257,-63.554,-177.709,7.308,148.708
C09839=1162.597,224.009,-63.529,-177.712,7.305,148.709
C09840=1162.601,223.760,-63.503,-177.714,7.303,148.709
C09841=1162.606,223.512,-63.478,-177.717,7.300,148.709
C09842=1162.611,223.263,-63.452,-177.719,7.298,148.709
C09843=1162.615,223.014,-63.426,-177.722,7.295,148.709
C09844=1162.620,222.766,-63.401,-177.725,7.293,148.709
C09845=1162.624,222.517,-63.376,-177.728,7.290,148.710
C09846=1162.628,222.268,-63.350,-177.730,7.287,148.710
C09847=1162.633,222.020,-63.325,-177.733,7.286,148.710
C09848=1162.637,221.771,-63.299,-177.736,7.283,148.710
C09849=1162.642,221.522,-63.274,-177.739,7.281,148.710
C09850=1162.647,221.273,-63.249,-177.741,7.278,148.711
C09851=1162.651,221.024,-63.223,-177.745,7.275,148.711
C09852=1162.656,220.776,-63.198,-177.747,7.273,148.711
C09853=1162.660,220.527,-63.172,-177.750,7.270,148.711
C09854=1162.664,220.279,-63.148,-177.752,7.269,148.711
C09855=1162.669,220.030,-63.123,-177.755,7.266,148.711
C09856=1162.674,219.782,-63.097,-177.758,7.264,148.712
C09857=1162.678,219.533,-63.072,-177.760,7.261,148.712
C09858=1162.683,219.283,-63.046,-177.763,7.259,148.712
C09859=1162.687,219.035,-63.021,-177.766,7.256,148.712
C09860=1162.691,218.786,-62.997,-177.769,7.253,148.712
C09861=1162.696,218.538,-62.971,-177.771,7.251,148.713
C09862=1162.700,218.289,-62.946,-177.774,7.249,148.713
C09863=1162.705,218.041,-62.921,-177.777,7.247,148.713
C09864=1162.710,217.792,-62.895,-177.780,7.244,148.713
C09865=1162.715,217.543,-62.870,-177.782,7.242,148.714
C09866=1162.718,217.295,-62.845,-177.785,7.239,148.714
C09867=1162.723,217.046,-62.821,-177.788,7.237,148.714
C09868=1162.728,216.797,-62.795,-177.790,7.234,148.714
C09869=1162.733,216.548,-62.770,-177.793,7.232,148.714
C09870=1162.736,216.300,-62.745,-177.796,7.230,148.715
C09871=1162.741,216.051,-62.720,-177.799,7.227,148.715
C09872=1162.745,215.802,-62.695,-177.801,7.225,148.715
C09873=1162.751,215.554,-62.670,-177.804,7.222,148.715
C09874=1162.754,215.304,-62.645,-177.807,7.220,148.715
C09875=1162.759,215.056,-62.620,-177.810,7.217,148.715
C09876=1162.764,214.807,-62.595,-177.812,7.216,148.716
C09877=1162.768,214.559,-62.570,-177.815,7.213,148.716
C09878=1162.772,214.310,-62.545,-177.818,7.211,148.716
C09879=1162.778,214.061,-62.521,-177.820,7.208,148.716
C09880=1162.781,213.812,-62.495,-177.823,7.206,148.717
C09881=1162.786,213.564,-62.471,-177.826,7.203,148.717
C09882=1162.791,213.315,-62.446,-177.829,7.201,148.717
C09883=1162.795,213.067,-62.421,-177.831,7.198,148.717
C09884=1162.800,212.818,-62.396,-177.834,7.197,148.718
C09885=1162.804,212.568,-62.371,-177.837,7.194,148.718
C09886=1162.809,212.320,-62.347,-177.839,7.192,148.718
C09887=1162.814,212.072,-62.322,-177.842,7.189,148.718
C09888=1162.817,211.823,-62.297,-177.845,7.187,148.718
C09889=1162.823,211.574,-62.273,-177.848,7.184,148.719
C09890=1162.827,211.325,-62.248,-177.850,7.183,148.719
C09891=1162.831,211.077,-62.223,-177.853,7.180,148.719
C09892=1162.836,210.828,-62.198,-177.856,7.178,148.719
C09893=1162.840,210.579,-62.174,-177.859,7.175,148.719
C09894=1162.845,210.309,-62.147,-177.862,7.172,148.720
C09895=1162.850,210.038,-62.120,-177.864,7.170,148.720
C09896=1162.855,209.768,-62.093,-177.867,7.168,148.720
C09897=1162.860,209.498,-62.067,-177.870,7.165,148.720
C09898=1162.865,209.248,-62.041,-177.873,7.163,148.721
C09899=1162.869,209.000,-62.017,-177.876,7.160,148.721
C09900=1162.874,208.751,-61.993,-177.878,7.158,148.721
C09901=1162.878,208.502,-61.968,-177.881,7.156,148.721
C09902=1162.883,208.253,-61.944,-177.884,7.153,148.721
C09903=1162.887,208.005,-61.920,-177.887,7.151,148.722
C09904=1162.892,207.755,-61.895,-177.889,7.149,148.722
C09905=1162.896,207.507,-61.870,-177.892,7.146,148.722
C09906=1162.902,207.258,-61.846,-177.894,7.144,148.722
C09907=1162.905,207.009,-61.821,-177.898,7.141,148.723
C09908=1162.910,206.760,-61.797,-177.900,7.139,148.723
C09909=1162.915,206.512,-61.773,-177.903,7.137,148.723
C09910=1162.920,206.263,-61.748,-177.906,7.135,148.723
C09911=1162.924,206.014,-61.723,-177.908,7.133,148.724
C09912=1162.928,205.766,-61.699,-177.911,7.130,148.724
C09913=1162.933,205.517,-61.675,-177.914,7.128,148.724
C09914=1162.937,205.268,-61.650,-177.917,7.126,148.724
C09915=1162.942,205.019,-61.626,-177.919,7.123,148.724
C09916=1162.947,204.771,-61.602,-177.922,7.121,148.725
C09917=1162.951,204.522,-61.577,-177.924,7.119,148.725
C09918=1162.956,204.272,-61.553,-177.928,7.116,148.725
C09919=1162.960,204.024,-61.529,-177.930,7.114,148.726
C09920=1162.965,203.775,-61.505,-177.933,7.112,148.726
C09921=1162.970,203.527,-61.480,-177.936,7.110,148.726
C09922=1162.974,203.278,-61.456,-177.938,7.108,148.726
C09923=1162.978,203.029,-61.432,-177.941,7.105,148.726
C09924=1162.983,202.780,-61.408,-177.943,7.103,148.727
C09925=1162.988,202.531,-61.384,-177.947,7.100,148.727
C09926=1162.992,202.283,-61.360,-177.949,7.099,148.727
C09927=1162.997,202.034,-61.335,-177.952,7.096,148.727
C09928=1163.001,201.785,-61.311,-177.955,7.094,148.728
C09929=1163.006,201.536,-61.287,-177.957,7.092,148.728
C09930=1163.010,201.288,-61.263,-177.960,7.089,148.728
C09931=1163.015,201.039,-61.238,-177.963,7.087,148.729
C09932=1163.019,200.789,-61.215,-177.966,7.084,148.729
C09933=1163.024,200.541,-61.191,-177.968,7.083,148.729
C09934=1163.028,200.292,-61.167,-177.971,7.081,148.729
C09935=1163.034,200.043,-61.143,-177.974,7.078,148.729
C09936=1163.038,199.795,-61.119,-177.977,7.076,148.730
C09937=1163.042,199.546,-61.095,-177.979,7.073,148.730
C09938=1163.047,199.297,-61.071,-177.982,7.072,148.730
C09939=1163.051,199.048,-61.047,-177.985,7.069,148.730
C09940=1163.056,198.799,-61.022,-177.987,7.067,148.731
C09941=1163.061,198.550,-60.999,-177.990,7.065,148.731
C09942=1163.065,198.302,-60.975,-177.993,7.062,148.731
C09943=1163.070,198.053,-60.951,-177.996,7.060,148.731
C09944=1163.074,197.805,-60.927,-177.998,7.057,148.732
C09945=1163.079,197.556,-60.904,-178.001,7.056,148.732
C09946=1163.083,197.307,-60.880,-178.004,7.054,148.732
C09947=1163.088,197.057,-60.855,-178.007,7.051,148.732
C09948=1163.093,196.809,-60.831,-178.009,7.049,148.733
C09949=1163.097,196.560,-60.808,-178.012,7.047,148.733
C09950=1163.102,196.311,-60.784,-178.015,7.044,148.733
C09951=1163.106,196.062,-60.761,-178.017,7.043,148.734
C09952=1163.111,195.814,-60.736,-178.021,7.040,148.734
C09953=1163.115,195.565,-60.713,-178.023,7.038,148.734
C09954=1163.120,195.316,-60.689,-178.025,7.036,148.734
C09955=1163.125,195.067,-60.666,-178.028,7.033,148.734
C09956=1163.129,194.819,-60.642,-178.031,7.032,148.735
C09957=1163.134,194.570,-60.618,-178.034,7.030,148.735
C09958=1163.138,194.321,-60.595,-178.036,7.027,148.735
C09959=1163.143,194.072,-60.571,-178.039,7.025,148.736
C09960=1163.148,193.823,-60.547,-178.042,7.023,148.736
C09961=1163.153,193.574,-60.524,-178.045,7.020,148.736
C09962=1163.157,193.326,-60.499,-178.047,7.019,148.736
C09963=1163.162,193.077,-60.476,-178.050,7.016,148.737
C09964=1163.167,192.828,-60.453,-178.053,7.014,148.737
C09965=1163.171,192.579,-60.429,-178.055,7.012,148.737
C09966=1163.176,192.330,-60.405,-178.059,7.010,148.738
C09967=1163.180,192.081,-60.383,-178.061,7.007,148.738
C09968=1163.184,191.833,-60.358,-178.064,7.006,148.738
C09969=1163.189,191.584,-60.335,-178.067,7.003,148.738
C09970=1163.194,191.335,-60.312,-178.069,7.001,148.739
C09971=1163.198,191.086,-60.288,-178.072,6.998,148.739
C09972=1163.203,190.837,-60.264,-178.075,6.997,148.739
C09973=1163.207,190.588,-60.241,-178.077,6.995,148.739
C09974=1163.212,190.339,-60.218,-178.080,6.992,148.740
C09975=1163.217,190.090,-60.194,-178.083,6.990,148.740
C09976=1163.221,189.841,-60.171,-178.085,6.988,148.740
C09977=1163.226,189.592,-60.148,-178.089,6.986,148.741
C09978=1163.231,189.344,-60.123,-178.091,6.984,148.741
C09979=1163.235,189.095,-60.100,-178.094,6.982,148.741
C09980=1163.239,188.846,-60.077,-178.097,6.979,148.741
C09981=1163.244,188.597,-60.054,-178.099,6.977,148.742
C09982=1163.249,188.348,-60.031,-178.102,6.976,148.742
C09983=1163.253,188.099,-60.007,-178.105,6.973,148.742
C09984=1163.258,187.850,-59.984,-178.108,6.971,148.743
C09985=1163.263,187.602,-59.961,-178.110,6.969,148.743
C09986=1163.267,187.353,-59.938,-178.113,6.966,148.743
C09987=1163.272,187.104,-59.915,-178.116,6.964,148.743
C09988=1163.277,186.855,-59.891,-178.118,6.963,148.744
C09989=1163.281,186.606,-59.868,-178.121,6.961,148.744
C09990=1163.286,186.357,-59.845,-178.124,6.958,148.744
C09991=1163.290,186.108,-59.822,-178.126,6.956,148.745
C09992=1163.295,185.859,-59.799,-178.129,6.954,148.745
C09993=1163.299,185.610,-59.775,-178.132,6.952,148.745
C09994=1163.305,185.362,-59.752,-178.135,6.950,148.745
C09995=1163.309,185.113,-59.729,-178.137,6.948,148.746
C09996=1163.313,184.864,-59.706,-178.141,6.945,148.746
//INST
///DATE 2021/06/25 14:30
///ATTR SC,RW,RJ
////FRAME ROBOT
///GROUP1 RB1
NOP
MOVL C00000 V=800.0 PL=0
MOVL C00001 V=800.0 PL=0
MOVL C00002 V=800.0 PL=0
MOVL C00003 V=800.0 PL=0
MOVL C00004 V=800.0 PL=0
MOVL C00005 V=800.0 PL=0
MOVL C00006 V=800.0 PL=0
MOVL C00007 V=800.0 PL=0
MOVL C00008 V=800.0 PL=0
MOVL C00009 V=800.0 PL=0
MOVL C00010 V=800.0 PL=0
MOVL C00011 V=800.0 PL=0
MOVL C00012 V=800.0 PL=0
MOVL C00013 V=800.0 PL=0
MOVL C00014 V=800.0 PL=0
MOVL C00015 V=800.0 PL=0
MOVL C00016 V=800.0 PL=0
MOVL C00017 V=800.0 PL=0
MOVL C00018 V=800.0 PL=0
MOVL C00019 V=800.0 PL=0
MOVL C00020 V=800.0 PL=0
MOVL C00021 V=800.0 PL=0
MOVL C00022 V=800.0 PL=0
MOVL C00023 V=800.0 PL=0
MOVL C00024 V=800.0 PL=0
MOVL C00025 V=800.0 PL=0
MOVL C00026 V=800.0 PL=0
MOVL C00027 V=800.0 PL=0
MOVL C00028 V=800.0 PL=0
MOVL C00029 V=800.0 PL=0
MOVL C00030 V=800.0 PL=0
MOVL C00031 V=800.0 PL=0
MOVL C00032 V=800.0 PL=0
MOVL C00033 V=800.0 PL=0
MOVL C00034 V=800.0 PL=0
MOVL C00035 V=800.0 PL=0
MOVL C00036 V=800.0 PL=0
MOVL C00037 V=800.0 PL=0
MOVL C00038 V=800.0 PL=0
MOVL C00039 V=800.0 PL=0
MOVL C00040 V=800.0 PL=0
MOVL C00041 V=800.0 PL=0
MOVL C00042 V=800.0 PL=0
MOVL C00043 V=800.0 PL=0
MOVL C00044 V=800.0 PL=0
MOVL C00045 V=800.0 PL=0
MOVL C00046 V=800.0 PL=0
MOVL C00047 V=800.0 PL=0
MOVL C00048 V=800.0 PL=0
MOVL C00049 V=800.0 PL=0
MOVL C00050 V=800.0 PL=0
MOVL C00051 V=800.0 PL=0
MOVL C00052 V=800.0 PL=0
MOVL C00053 V=800.0 PL=0
MOVL C00054 V=800.0 PL=0
MOVL C00055 V=800.0 PL=0
MOVL C00056 V=800.0 PL=0
MOVL C00057 V=800.0 PL=0
MOVL C00058 V=800.0 PL=0
MOVL C00059 V=800.0 PL=0
MOVL C00060 V=800.0 PL=0
MOVL C00061 V=800.0 PL=0
MOVL C00062 V=800.0 PL=0
MOVL C00063 V=800.0 PL=0
MOVL C00064 V=800.0 PL=0
MOVL C00065 V=800.0 PL=0
MOVL C00066 V=800.0 PL=0
MOVL C00067 V=800.0 PL=0
MOVL C00068 V=800.0 PL=0
MOVL C00069 V=800.0 PL=0
MOVL C00070 V=800.0 PL=0
MOVL C00071 V=800.0 PL=0
MOVL C00072 V=800.0 PL=0
MOVL C00073 V=800.0 PL=0
MOVL C00074 V=800.0 PL=0
MOVL C00075 V=800.0 PL=0
MOVL C00076 V=800.0 PL=0
MOVL C00077 V=800.0 PL=0
MOVL C00078 V=800.0 PL=0
MOVL C00079 V=800.0 PL=0
MOVL C00080 V=800.0 PL=0
MOVL C00081 V=800.0 PL=0
MOVL C00082 V=800.0 PL=0
MOVL C00083 V=800.0 PL=0
MOVL C00084 V=800.0 PL=0
MOVL C00085 V=800.0 PL=0
MOVL C00086 V=800.0 PL=0
MOVL C00087 V=800.0 PL=0
MOVL C00088 V=800.0 PL=0
MOVL C00089 V=800.0 PL=0
MOVL C00090 V=800.0 PL=0
MOVL C00091 V=800.0 PL=0
MOVL C00092 V=800.0 PL=0
MOVL C00093 V=800.0 PL=0
MOVL C00094 V=800.0 PL=0
MOVL C00095 V=800.0 PL=0
MOVL C00096 V=800.0 PL=0
MOVL C00097 V=800.0 PL=0
MOVL C00098 V=800.0 PL=0
MOVL C00099 V=800.0 PL=0
MOVL C00100 V=800.0 PL=0
MOVL C00101 V=800.0 PL=0
MOVL C00102 V=800.0 PL=0
MOVL C00103 V=800.0 PL=0
MOVL C00104 V=800.0 PL=0
MOVL C00105 V=800.0 PL=0
MOVL C00106 V=800.0 PL=0
MOVL C00107 V=800.0 PL=0
MOVL C00108 V=800.0 PL=0
MOVL C00109 V=800.0 PL=0
MOVL C00110 V=800.0 PL=0
MOVL C00111 V=800.0 PL=0
MOVL C00112 V=800.0 PL=0
MOVL C00113 V=800.0 PL=0
MOVL C00114 V=800.0 PL=0
MOVL C00115 V=800.0 PL=0
MOVL C00116 V=800.0 PL=0
MOVL C00117 V=800.0 PL=0
MOVL C00118 V=800.0 PL=0
MOVL C00119 V=800.0 PL=0
MOVL C00120 V=800.0 PL=0
MOVL C00121 V=800.0 PL=0
MOVL C00122 V=800.0 PL=0
MOVL C00123 V=800.0 PL=0
MOVL C00124 V=800.0 PL=0
MOVL C00125 V=800.0 PL=0
MOVL C00126 V=800.0 PL=0
MOVL C00127 V=800.0 PL=0
MOVL C00128 V=800.0 PL=0
MOVL C00129 V=800.0 PL=0
MOVL C00130 V=800.0 PL=0
MOVL C00131 V=800.0 PL=0
MOVL C00132 V=800.0 PL=0
MOVL C00133 V=800.0 PL=0
MOVL C00134 V=800.0 PL=0
MOVL C00135 V=800.0 PL=0
MOVL C00136 V=800.0 PL=0
MOVL C00137 V=800.0 PL=0
MOVL C00138 V=800.0 PL=0
MOVL C00139 V=800.0 PL=0
MOVL C00140 V=800.0 PL=0
MOVL C00141 V=800.0 PL=0
MOVL C00142 V=800.0 PL=0
MOVL C00143 V=800.0 PL=0
MOVL C00144 V=800.0 PL=0
MOVL C00145 V=800.0 PL=0
MOVL C00146 V=800.0 PL=0
MOVL C00147 V=800.0 PL=0
MOVL C00148 V=800.0 PL=0
MOVL C00149 V=800.0 PL=0
MOVL C00150 V=800.0 PL=0
MOVL C00151 V=800.0 PL=0
MOVL C00152 V=800.0 PL=0
MOVL C00153 V=800.0 PL=0
MOVL C00154 V=800.0 PL=0
MOVL C00155 V=800.0 PL=0
MOVL C00156 V=800.0 PL=0
MOVL C00157 V=800.0 PL=0
MOVL C00158 V=800.0 PL=0
MOVL C00159 V=800.0 PL=0
MOVL C00160 V=800.0 PL=0
MOVL C00161 V=800.0 PL=0
MOVL C00162 V=800.0 PL=0
MOVL C00163 V=800.0 PL=0
MOVL C00164 V=800.0 PL=0
MOVL C00165 V=800.0 PL=0
MOVL C00166 V=800.0 PL=0
MOVL C00167 V=800.0 PL=0
MOVL C00168 V=800.0 PL=0
MOVL C00169 V=800.0 PL=0
MOVL C00170 V=800.0 PL=0
MOVL C00171 V=800.0 PL=0
MOVL C00172 V=800.0 PL=0
MOVL C00173 V=800.0 PL=0
MOVL C00174 V=800.0 PL=0
MOVL C00175 V=800.0 PL=0
MOVL C00176 V=800.0 PL=0
MOVL C00177 V=800.0 PL=0
MOVL C00178 V=800.0 PL=0
MOVL C00179 V=800.0 PL=0
MOVL C00180 V=800.0 PL=0
MOVL C00181 V=800.0 PL=0
MOVL C00182 V=800.0 PL=0
MOVL C00183 V=800.0 PL=0
MOVL C00184 V=800.0 PL=0
MOVL C00185 V=800.0 PL=0
MOVL C00186 V=800.0 PL=0
MOVL C00187 V=800.0 PL=0
MOVL C00188 V=800.0 PL=0
MOVL C00189 V=800.0 PL=0
MOVL C00190 V=800.0 PL=0
MOVL C00191 V=800.0 PL=0
MOVL C00192 V=800.0 PL=0
MOVL C00193 V=800.0 PL=0
MOVL C00194 V=800.0 PL=0
MOVL C00195 V=800.0 PL=0
MOVL C00196 V=800.0 PL=0
MOVL C00197 V=800.0 PL=0
MOVL C00198 V=800.0 PL=0
MOVL C00199 V=800.0 PL=0
MOVL C00200 V=800.0 PL=0
MOVL C00201 V=800.0 PL=0
MOVL C00202 V=800.0 PL=0
MOVL C00203 V=800.0 PL=0
MOVL C00204 V=800.0 PL=0
MOVL C00205 V=800.0 PL=0
MOVL C00206 V=800.0 PL=0
MOVL C00207 V=800.0 PL=0
MOVL C00208 V=800.0 PL=0
MOVL C00209 V=800.0 PL=0
MOVL C00210 V=800.0 PL=0
MOVL C00211 V=800.0 PL=0
MOVL C00212 V=800.0 PL=0
MOVL C00213 V=800.0 PL=0
MOVL C00214 V=800.0 PL=0
MOVL C00215 V=800.0 PL=0
MOVL C00216 V=800.0 PL=0
MOVL C00217 V=800.0 PL=0
MOVL C00218 V=800.0 PL=0
MOVL C00219 V=800.0 PL=0
MOVL C00220 V=800.0 PL=0
MOVL C00221 V=800.0 PL=0
MOVL C00222 V=800.0 PL=0
MOVL C00223 V=800.0 PL=0
MOVL C00224 V=800.0 PL=0
MOVL C00225 V=800.0 PL=0
MOVL C00226 V=800.0 PL=0
MOVL C00227 V=800.0 PL=0
MOVL C00228 V=800.0 PL=0
MOVL C00229 V=800.0 PL=0
MOVL C00230 V=800.0 PL=0
MOVL C00231 V=800.0 PL=0
MOVL C00232 V=800.0 PL=0
MOVL C00233 V=800.0 PL=0
MOVL C00234 V=800.0 PL=0
MOVL C00235 V=800.0 PL=0
MOVL C00236 V=800.0 PL=0
MOVL C00237 V=800.0 PL=0
MOVL C00238 V=800.0 PL=0
MOVL C00239 V=800.0 PL=0
MOVL C00240 V=800.0 PL=0
MOVL C00241 V=800.0 PL=0
MOVL C00242 V=800.0 PL=0
MOVL C00243 V=800.0 PL=0
MOVL C00244 V=800.0 PL=0
MOVL C00245 V=800.0 PL=0
MOVL C00246 V=800.0 PL=0
MOVL C00247 V=800.0 PL=0
MOVL C00248 V=800.0 PL=0
MOVL C00249 V=800.0 PL=0
MOVL C00250 V=800.0 PL=0
MOVL C00251 V=800.0 PL=0
MOVL C00252 V=800.0 PL=0
MOVL C00253 V=800.0 PL=0
MOVL C00254 V=800.0 PL=0
MOVL C00255 V=800.0 PL=0
MOVL C00256 V=800.0 PL=0
MOVL C00257 V=800.0 PL=0
MOVL C00258 V=800.0 PL=0
MOVL C00259 V=800.0 PL=0
MOVL C00260 V=800.0 PL=0
MOVL C00261 V=800.0 PL=0
MOVL C00262 V=800.0 PL=0
MOVL C00263 V=800.0 PL=0
MOVL C00264 V=800.0 PL=0
MOVL C00265 V=800.0 PL=0
MOVL C00266 V=800.0 PL=0
MOVL C00267 V=800.0 PL=0
MOVL C00268 V=800.0 PL=0
MOVL C00269 V=800.0 PL=0
MOVL C00270 V=800.0 PL=0
MOVL C00271 V=800.0 PL=0
MOVL C00272 V=800.0 PL=0
MOVL C00273 V=800.0 PL=0
MOVL C00274 V=800.0 PL=0
MOVL C00275 V=800.0 PL=0
MOVL C00276 V=800.0 PL=0
MOVL C00277 V=800.0 PL=0
MOVL C00278 V=800.0 PL=0
MOVL C00279 V=800.0 PL=0
MOVL C00280 V=800.0 PL=0
MOVL C00281 V=800.0 PL=0
MOVL C00282 V=800.0 PL=0
MOVL C00283 V=800.0 PL=0
MOVL C00284 V=800.0 PL=0
MOVL C00285 V=800.0 PL=0
MOVL C00286 V=800.0 PL=0
MOVL C00287 V=800.0 PL=0
MOVL C00288 V=800.0 PL=0
MOVL C00289 V=800.0 PL=0
MOVL C00290 V=800.0 PL=0
MOVL C00291 V=800.0 PL=0
MOVL C00292 V=800.0 PL=0
MOVL C00293 V=800.0 PL=0
MOVL C00294 V=800.0 PL=0
MOVL C00295 V=800.0 PL=0
MOVL C00296 V=800.0 PL=0
MOVL C00297 V=800.0 PL=0
MOVL C00298 V=800.0 PL=0
MOVL C00299 V=800.0 PL=0
MOVL C00300 V=800.0 PL=0
MOVL C00301 V=800.0 PL=0
MOVL C00302 V=800.0 PL=0
MOVL C00303 V=800.0 PL=0
MOVL C00304 V=800.0 PL=0
MOVL C00305 V=800.0 PL=0
MOVL C00306 V=800.0 PL=0
MOVL C00307 V=800.0 PL=0
MOVL C00308 V=800.0 PL=0
MOVL C00309 V=800.0 PL=0
MOVL C00310 V=800.0 PL=0
MOVL C00311 V=800.0 PL=0
MOVL C00312 V=800.0 PL=0
MOVL C00313 V=800.0 PL=0
MOVL C00314 V=800.0 PL=0
MOVL C00315 V=800.0 PL=0
MOVL C00316 V=800.0 PL=0
MOVL C00317 V=800.0 PL=0
MOVL C00318 V=800.0 PL=0
MOVL C00319 V=800.0 PL=0
MOVL C00320 V=800.0 PL=0
MOVL C00321 V=800.0 PL=0
MOVL C00322 V=800.0 PL=0
MOVL C00323 V=800.0 PL=0
MOVL C00324 V=800.0 PL=0
MOVL C00325 V=800.0 PL=0
MOVL C00326 V=800.0 PL=0
MOVL C00327 V=800.0 PL=0
MOVL C00328 V=800.0 PL=0
MOVL C00329 V=800.0 PL=0
MOVL C00330 V=800.0 PL=0
MOVL C00331 V=800.0 PL=0
MOVL C00332 V=800.0 PL=0
MOVL C00333 V=800.0 PL=0
MOVL C00334 V=800.0 PL=0
MOVL C00335 V=800.0 PL=0
MOVL C00336 V=800.0 PL=0
MOVL C00337 V=800.0 PL=0
MOVL C00338 V=800.0 PL=0
MOVL C00339 V=800.0 PL=0
MOVL C00340 V=800.0 PL=0
MOVL C00341 V=800.0 PL=0
MOVL C00342 V=800.0 PL=0
MOVL C00343 V=800.0 PL=0
MOVL C00344 V=800.0 PL=0
MOVL C00345 V=800.0 PL=0
MOVL C00346 V=800.0 PL=0
MOVL C00347 V=800.0 PL=0
MOVL C00348 V=800.0 PL=0
MOVL C00349 V=800.0 PL=0
MOVL C00350 V=800.0 PL=0
MOVL C00351 V=800.0 PL=0
MOVL C00352 V=800.0 PL=0
MOVL C00353 V=800.0 PL=0
MOVL C00354 V=800.0 PL=0
MOVL C00355 V=800.0 PL=0
MOVL C00356 V=800.0 PL=0
MOVL C00357 V=800.0 PL=0
MOVL C00358 V=800.0 PL=0
MOVL C00359 V=800.0 PL=0
MOVL C00360 V=800.0 PL=0
MOVL C00361 V=800.0 PL=0
MOVL C00362 V=800.0 PL=0
MOVL C00363 V=800.0 PL=0
MOVL C00364 V=800.0 PL=0
MOVL C00365 V=800.0 PL=0
MOVL C00366 V=800.0 PL=0
MOVL C00367 V=800.0 PL=0
MOVL C00368 V=800.0 PL=0
MOVL C00369 V=800.0 PL=0
MOVL C00370 V=800.0 PL=0
MOVL C00371 V=800.0 PL=0
MOVL C00372 V=800.0 PL=0
MOVL C00373 V=800.0 PL=0
MOVL C00374 V=800.0 PL=0
MOVL C00375 V=800.0 PL=0
MOVL C00376 V=800.0 PL=0
MOVL C00377 V=800.0 PL=0
MOVL C00378 V=800.0 PL=0
MOVL C00379 V=800.0 PL=0
MOVL C00380 V=800.0 PL=0
MOVL C00381 V=800.0 PL=0
MOVL C00382 V=800.0 PL=0
MOVL C00383 V=800.0 PL=0
MOVL C00384 V=800.0 PL=0
MOVL C00385 V=800.0 PL=0
MOVL C00386 V=800.0 PL=0
MOVL C00387 V=800.0 PL=0
MOVL C00388 V=800.0 PL=0
MOVL C00389 V=800.0 PL=0
MOVL C00390 V=800.0 PL=0
MOVL C00391 V=800.0 PL=0
MOVL C00392 V=800.0 PL=0
MOVL C00393 V=800.0 PL=0
MOVL C00394 V=800.0 PL=0
MOVL C00395 V=800.0 PL=0
MOVL C00396 V=800.0 PL=0
MOVL C00397 V=800.0 PL=0
MOVL C00398 V=800.0 PL=0
MOVL C00399 V=800.0 PL=0
MOVL C00400 V=800.0 PL=0
MOVL C00401 V=800.0 PL=0
MOVL C00402 V=800.0 PL=0
MOVL C00403 V=800.0 PL=0
MOVL C00404 V=800.0 PL=0
MOVL C00405 V=800.0 PL=0
MOVL C00406 V=800.0 PL=0
MOVL C00407 V=800.0 PL=0
MOVL C00408 V=800.0 PL=0
MOVL C00409 V=800.0 PL=0
MOVL C00410 V=800.0 PL=0
MOVL C00411 V=800.0 PL=0
MOVL C00412 V=800.0 PL=0
MOVL C00413 V=800.0 PL=0
MOVL C00414 V=800.0 PL=0
MOVL C00415 V=800.0 PL=0
MOVL C00416 V=800.0 PL=0
MOVL C00417 V=800.0 PL=0
MOVL C00418 V=800.0 PL=0
MOVL C00419 V=800.0 PL=0
MOVL C00420 V=800.0 PL=0
MOVL C00421 V=800.0 PL=0
MOVL C00422 V=800.0 PL=0
MOVL C00423 V=800.0 PL=0
MOVL C00424 V=800.0 PL=0
MOVL C00425 V=800.0 PL=0
MOVL C00426 V=800.0 PL=0
MOVL C00427 V=800.0 PL=0
MOVL C00428 V=800.0 PL=0
MOVL C00429 V=800.0 PL=0
MOVL C00430 V=800.0 PL=0
MOVL C00431 V=800.0 PL=0
MOVL C00432 V=800.0 PL=0
MOVL C00433 V=800.0 PL=0
MOVL C00434 V=800.0 PL=0
MOVL C00435 V=800.0 PL=0
MOVL C00436 V=800.0 PL=0
MOVL C00437 V=800.0 PL=0
MOVL C00438 V=800.0 PL=0
MOVL C00439 V=800.0 PL=0
MOVL C00440 V=800.0 PL=0
MOVL C00441 V=800.0 PL=0
MOVL C00442 V=800.0 PL=0
MOVL C00443 V=800.0 PL=0
MOVL C00444 V=800.0 PL=0
MOVL C00445 V=800.0 PL=0
MOVL C00446 V=800.0 PL=0
MOVL C00447 V=800.0 PL=0
MOVL C00448 V=800.0 PL=0
MOVL C00449 V=800.0 PL=0
MOVL C00450 V=800.0 PL=0
MOVL C00451 V=800.0 PL=0
MOVL C00452 V=800.0 PL=0
MOVL C00453 V=800.0 PL=0
MOVL C00454 V=800.0 PL=0
MOVL C00455 V=800.0 PL=0
MOVL C00456 V=800.0 PL=0
MOVL C00457 V=800.0 PL=0
MOVL C00458 V=800.0 PL=0
MOVL C00459 V=800.0 PL=0
MOVL C00460 V=800.0 PL=0
MOVL C00461 V=800.0 PL=0
MOVL C00462 V=800.0 PL=0
MOVL C00463 V=800.0 PL=0
MOVL C00464 V=800.0 PL=0
MOVL C00465 V=800.0 PL=0
MOVL C00466 V=800.0 PL=0
MOVL C00467 V=800.0 PL=0
MOVL C00468 V=800.0 PL=0
MOVL C00469 V=800.0 PL=0
MOVL C00470 V=800.0 PL=0
MOVL C00471 V=800.0 PL=0
MOVL C00472 V=800.0 PL=0
MOVL C00473 V=800.0 PL=0
MOVL C00474 V=800.0 PL=0
MOVL C00475 V=800.0 PL=0
MOVL C00476 V=800.0 PL=0
MOVL C00477 V=800.0 PL=0
MOVL C00478 V=800.0 PL=0
MOVL C00479 V=800.0 PL=0
MOVL C00480 V=800.0 PL=0
MOVL C00481 V=800.0 PL=0
MOVL C00482 V=800.0 PL=0
MOVL C00483 V=800.0 PL=0
MOVL C00484 V=800.0 PL=0
MOVL C00485 V=800.0 PL=0
MOVL C00486 V=800.0 PL=0
MOVL C00487 V=800.0 PL=0
MOVL C00488 V=800.0 PL=0
MOVL C00489 V=800.0 PL=0
MOVL C00490 V=800.0 PL=0
MOVL C00491 V=800.0 PL=0
MOVL C00492 V=800.0 PL=0
MOVL C00493 V=800.0 PL=0
MOVL C00494 V=800.0 PL=0
MOVL C00495 V=800.0 PL=0
MOVL C00496 V=800.0 PL=0
MOVL C00497 V=800.0 PL=0
MOVL C00498 V=800.0 PL=0
MOVL C00499 V=800.0 PL=0
MOVL C00500 V=800.0 PL=0
MOVL C00501 V=800.0 PL=0
MOVL C00502 V=800.0 PL=0
MOVL C00503 V=800.0 PL=0
MOVL C00504 V=800.0 PL=0
MOVL C00505 V=800.0 PL=0
MOVL C00506 V=800.0 PL=0
MOVL C00507 V=800.0 PL=0
MOVL C00508 V=800.0 PL=0
MOVL C00509 V=800.0 PL=0
MOVL C00510 V=800.0 PL=0
MOVL C00511 V=800.0 PL=0
MOVL C00512 V=800.0 PL=0
MOVL C00513 V=800.0 PL=0
MOVL C00514 V=800.0 PL=0
MOVL C00515 V=800.0 PL=0
MOVL C00516 V=800.0 PL=0
MOVL C00517 V=800.0 PL=0
MOVL C00518 V=800.0 PL=0
MOVL C00519 V=800.0 PL=0
MOVL C00520 V=800.0 PL=0
MOVL C00521 V=800.0 PL=0
MOVL C00522 V=800.0 PL=0
MOVL C00523 V=800.0 PL=0
MOVL C00524 V=800.0 PL=0
MOVL C00525 V=800.0 PL=0
MOVL C00526 V=800.0 PL=0
MOVL C00527 V=800.0 PL=0
MOVL C00528 V=800.0 PL=0
MOVL C00529 V=800.0 PL=0
MOVL C00530 V=800.0 PL=0
MOVL C00531 V=800.0 PL=0
MOVL C00532 V=800.0 PL=0
MOVL C00533 V=800.0 PL=0
MOVL C00534 V=800.0 PL=0
MOVL C00535 V=800.0 PL=0
MOVL C00536 V=800.0 PL=0
MOVL C00537 V=800.0 PL=0
MOVL C00538 V=800.0 PL=0
MOVL C00539 V=800.0 PL=0
MOVL C00540 V=800.0 PL=0
MOVL C00541 V=800.0 PL=0
MOVL C00542 V=800.0 PL=0
MOVL C00543 V=800.0 PL=0
MOVL C00544 V=800.0 PL=0
MOVL C00545 V=800.0 PL=0
MOVL C00546 V=800.0 PL=0
MOVL C00547 V=800.0 PL=0
MOVL C00548 V=800.0 PL=0
MOVL C00549 V=800.0 PL=0
MOVL C00550 V=800.0 PL=0
MOVL C00551 V=800.0 PL=0
MOVL C00552 V=800.0 PL=0
MOVL C00553 V=800.0 PL=0
MOVL C00554 V=800.0 PL=0
MOVL C00555 V=800.0 PL=0
MOVL C00556 V=800.0 PL=0
MOVL C00557 V=800.0 PL=0
MOVL C00558 V=800.0 PL=0
MOVL C00559 V=800.0 PL=0
MOVL C00560 V=800.0 PL=0
MOVL C00561 V=800.0 PL=0
MOVL C00562 V=800.0 PL=0
MOVL C00563 V=800.0 PL=0
MOVL C00564 V=800.0 PL=0
MOVL C00565 V=800.0 PL=0
MOVL C00566 V=800.0 PL=0
MOVL C00567 V=800.0 PL=0
MOVL C00568 V=800.0 PL=0
MOVL C00569 V=800.0 PL=0
MOVL C00570 V=800.0 PL=0
MOVL C00571 V=800.0 PL=0
MOVL C00572 V=800.0 PL=0
MOVL C00573 V=800.0 PL=0
MOVL C00574 V=800.0 PL=0
MOVL C00575 V=800.0 PL=0
MOVL C00576 V=800.0 PL=0
MOVL C00577 V=800.0 PL=0
MOVL C00578 V=800.0 PL=0
MOVL C00579 V=800.0 PL=0
MOVL C00580 V=800.0 PL=0
MOVL C00581 V=800.0 PL=0
MOVL C00582 V=800.0 PL=0
MOVL C00583 V=800.0 PL=0
MOVL C00584 V=800.0 PL=0
MOVL C00585 V=800.0 PL=0
MOVL C00586 V=800.0 PL=0
MOVL C00587 V=800.0 PL=0
MOVL C00588 V=800.0 PL=0
MOVL C00589 V=800.0 PL=0
MOVL C00590 V=800.0 PL=0
MOVL C00591 V=800.0 PL=0
MOVL C00592 V=800.0 PL=0
MOVL C00593 V=800.0 PL=0
MOVL C00594 V=800.0 PL=0
MOVL C00595 V=800.0 PL=0
MOVL C00596 V=800.0 PL=0
MOVL C00597 V=800.0 PL=0
MOVL C00598 V=800.0 PL=0
MOVL C00599 V=800.0 PL=0
MOVL C00600 V=800.0 PL=0
MOVL C00601 V=800.0 PL=0
MOVL C00602 V=800.0 PL=0
MOVL C00603 V=800.0 PL=0
MOVL C00604 V=800.0 PL=0
MOVL C00605 V=800.0 PL=0
MOVL C00606 V=800.0 PL=0
MOVL C00607 V=800.0 PL=0
MOVL C00608 V=800.0 PL=0
MOVL C00609 V=800.0 PL=0
MOVL C00610 V=800.0 PL=0
MOVL C00611 V=800.0 PL=0
MOVL C00612 V=800.0 PL=0
MOVL C00613 V=800.0 PL=0
MOVL C00614 V=800.0 PL=0
MOVL C00615 V=800.0 PL=0
MOVL C00616 V=800.0 PL=0
MOVL C00617 V=800.0 PL=0
MOVL C00618 V=800.0 PL=0
MOVL C00619 V=800.0 PL=0
MOVL C00620 V=800.0 PL=0
MOVL C00621 V=800.0 PL=0
MOVL C00622 V=800.0 PL=0
MOVL C00623 V=800.0 PL=0
MOVL C00624 V=800.0 PL=0
MOVL C00625 V=800.0 PL=0
MOVL C00626 V=800.0 PL=0
MOVL C00627 V=800.0 PL=0
MOVL C00628 V=800.0 PL=0
MOVL C00629 V=800.0 PL=0
MOVL C00630 V=800.0 PL=0
MOVL C00631 V=800.0 PL=0
MOVL C00632 V=800.0 PL=0
MOVL C00633 V=800.0 PL=0
MOVL C00634 V=800.0 PL=0
MOVL C00635 V=800.0 PL=0
MOVL C00636 V=800.0 PL=0
MOVL C00637 V=800.0 PL=0
MOVL C00638 V=800.0 PL=0
MOVL C00639 V=800.0 PL=0
MOVL C00640 V=800.0 PL=0
MOVL C00641 V=800.0 PL=0
MOVL C00642 V=800.0 PL=0
MOVL C00643 V=800.0 PL=0
MOVL C00644 V=800.0 PL=0
MOVL C00645 V=800.0 PL=0
MOVL C00646 V=800.0 PL=0
MOVL C00647 V=800.0 PL=0
MOVL C00648 V=800.0 PL=0
MOVL C00649 V=800.0 PL=0
MOVL C00650 V=800.0 PL=0
MOVL C00651 V=800.0 PL=0
MOVL C00652 V=800.0 PL=0
MOVL C00653 V=800.0 PL=0
MOVL C00654 V=800.0 PL=0
MOVL C00655 V=800.0 PL=0
MOVL C00656 V=800.0 PL=0
MOVL C00657 V=800.0 PL=0
MOVL C00658 V=800.0 PL=0
MOVL C00659 V=800.0 PL=0
MOVL C00660 V=800.0 PL=0
MOVL C00661 V=800.0 PL=0
MOVL C00662 V=800.0 PL=0
MOVL C00663 V=800.0 PL=0
MOVL C00664 V=800.0 PL=0
MOVL C00665 V=800.0 PL=0
MOVL C00666 V=800.0 PL=0
MOVL C00667 V=800.0 PL=0
MOVL C00668 V=800.0 PL=0
MOVL C00669 V=800.0 PL=0
MOVL C00670 V=800.0 PL=0
MOVL C00671 V=800.0 PL=0
MOVL C00672 V=800.0 PL=0
MOVL C00673 V=800.0 PL=0
MOVL C00674 V=800.0 PL=0
MOVL C00675 V=800.0 PL=0
MOVL C00676 V=800.0 PL=0
MOVL C00677 V=800.0 PL=0
MOVL C00678 V=800.0 PL=0
MOVL C00679 V=800.0 PL=0
MOVL C00680 V=800.0 PL=0
MOVL C00681 V=800.0 PL=0
MOVL C00682 V=800.0 PL=0
MOVL C00683 V=800.0 PL=0
MOVL C00684 V=800.0 PL=0
MOVL C00685 V=800.0 PL=0
MOVL C00686 V=800.0 PL=0
MOVL C00687 V=800.0 PL=0
MOVL C00688 V=800.0 PL=0
MOVL C00689 V=800.0 PL=0
MOVL C00690 V=800.0 PL=0
MOVL C00691 V=800.0 PL=0
MOVL C00692 V=800.0 PL=0
MOVL C00693 V=800.0 PL=0
MOVL C00694 V=800.0 PL=0
MOVL C00695 V=800.0 PL=0
MOVL C00696 V=800.0 PL=0
MOVL C00697 V=800.0 PL=0
MOVL C00698 V=800.0 PL=0
MOVL C00699 V=800.0 PL=0
MOVL C00700 V=800.0 PL=0
MOVL C00701 V=800.0 PL=0
MOVL C00702 V=800.0 PL=0
MOVL C00703 V=800.0 PL=0
MOVL C00704 V=800.0 PL=0
MOVL C00705 V=800.0 PL=0
MOVL C00706 V=800.0 PL=0
MOVL C00707 V=800.0 PL=0
MOVL C00708 V=800.0 PL=0
MOVL C00709 V=800.0 PL=0
MOVL C00710 V=800.0 PL=0
MOVL C00711 V=800.0 PL=0
MOVL C00712 V=800.0 PL=0
MOVL C00713 V=800.0 PL=0
MOVL C00714 V=800.0 PL=0
MOVL C00715 V=800.0 PL=0
MOVL C00716 V=800.0 PL=0
MOVL C00717 V=800.0 PL=0
MOVL C00718 V=800.0 PL=0
MOVL C00719 V=800.0 PL=0
MOVL C00720 V=800.0 PL=0
MOVL C00721 V=800.0 PL=0
MOVL C00722 V=800.0 PL=0
MOVL C00723 V=800.0 PL=0
MOVL C00724 V=800.0 PL=0
MOVL C00725 V=800.0 PL=0
MOVL C00726 V=800.0 PL=0
MOVL C00727 V=800.0 PL=0
MOVL C00728 V=800.0 PL=0
MOVL C00729 V=800.0 PL=0
MOVL C00730 V=800.0 PL=0
MOVL C00731 V=800.0 PL=0
MOVL C00732 V=800.0 PL=0
MOVL C00733 V=800.0 PL=0
MOVL C00734 V=800.0 PL=0
MOVL C00735 V=800.0 PL=0
MOVL C00736 V=800.0 PL=0
MOVL C00737 V=800.0 PL=0
MOVL C00738 V=800.0 PL=0
MOVL C00739 V=800.0 PL=0
MOVL C00740 V=800.0 PL=0
MOVL C00741 V=800.0 PL=0
MOVL C00742 V=800.0 PL=0
MOVL C00743 V=800.0 PL=0
MOVL C00744 V=800.0 PL=0
MOVL C00745 V=800.0 PL=0
MOVL C00746 V=800.0 PL=0
MOVL C00747 V=800.0 PL=0
MOVL C00748 V=800.0 PL=0
MOVL C00749 V=800.0 PL=0
MOVL C00750 V=800.0 PL=0
MOVL C00751 V=800.0 PL=0
MOVL C00752 V=800.0 PL=0
MOVL C00753 V=800.0 PL=0
MOVL C00754 V=800.0 PL=0
MOVL C00755 V=800.0 PL=0
MOVL C00756 V=800.0 PL=0
MOVL C00757 V=800.0 PL=0
MOVL C00758 V=800.0 PL=0
MOVL C00759 V=800.0 PL=0
MOVL C00760 V=800.0 PL=0
MOVL C00761 V=800.0 PL=0
MOVL C00762 V=800.0 PL=0
MOVL C00763 V=800.0 PL=0
MOVL C00764 V=800.0 PL=0
MOVL C00765 V=800.0 PL=0
MOVL C00766 V=800.0 PL=0
MOVL C00767 V=800.0 PL=0
MOVL C00768 V=800.0 PL=0
MOVL C00769 V=800.0 PL=0
MOVL C00770 V=800.0 PL=0
MOVL C00771 V=800.0 PL=0
MOVL C00772 V=800.0 PL=0
MOVL C00773 V=800.0 PL=0
MOVL C00774 V=800.0 PL=0
MOVL C00775 V=800.0 PL=0
MOVL C00776 V=800.0 PL=0
MOVL C00777 V=800.0 PL=0
MOVL C00778 V=800.0 PL=0
MOVL C00779 V=800.0 PL=0
MOVL C00780 V=800.0 PL=0
MOVL C00781 V=800.0 PL=0
MOVL C00782 V=800.0 PL=0
MOVL C00783 V=800.0 PL=0
MOVL C00784 V=800.0 PL=0
MOVL C00785 V=800.0 PL=0
MOVL C00786 V=800.0 PL=0
MOVL C00787 V=800.0 PL=0
MOVL C00788 V=800.0 PL=0
MOVL C00789 V=800.0 PL=0
MOVL C00790 V=800.0 PL=0
MOVL C00791 V=800.0 PL=0
MOVL C00792 V=800.0 PL=0
MOVL C00793 V=800.0 PL=0
MOVL C00794 V=800.0 PL=0
MOVL C00795 V=800.0 PL=0
MOVL C00796 V=800.0 PL=0
MOVL C00797 V=800.0 PL=0
MOVL C00798 V=800.0 PL=0
MOVL C00799 V=800.0 PL=0
MOVL C00800 V=800.0 PL=0
MOVL C00801 V=800.0 PL=0
MOVL C00802 V=800.0 PL=0
MOVL C00803 V=800.0 PL=0
MOVL C00804 V=800.0 PL=0
MOVL C00805 V=800.0 PL=0
MOVL C00806 V=800.0 PL=0
MOVL C00807 V=800.0 PL=0
MOVL C00808 V=800.0 PL=0
MOVL C00809 V=800.0 PL=0
MOVL C00810 V=800.0 PL=0
MOVL C00811 V=800.0 PL=0
MOVL C00812 V=800.0 PL=0
MOVL C00813 V=800.0 PL=0
MOVL C00814 V=800.0 PL=0
MOVL C00815 V=800.0 PL=0
MOVL C00816 V=800.0 PL=0
MOVL C00817 V=800.0 PL=0
MOVL C00818 V=800.0 PL=0
MOVL C00819 V=800.0 PL=0
MOVL C00820 V=800.0 PL=0
MOVL C00821 V=800.0 PL=0
MOVL C00822 V=800.0 PL=0
MOVL C00823 V=800.0 PL=0
MOVL C00824 V=800.0 PL=0
MOVL C00825 V=800.0 PL=0
MOVL C00826 V=800.0 PL=0
MOVL C00827 V=800.0 PL=0
MOVL C00828 V=800.0 PL=0
MOVL C00829 V=800.0 PL=0
MOVL C00830 V=800.0 PL=0
MOVL C00831 V=800.0 PL=0
MOVL C00832 V=800.0 PL=0
MOVL C00833 V=800.0 PL=0
MOVL C00834 V=800.0 PL=0
MOVL C00835 V=800.0 PL=0
MOVL C00836 V=800.0 PL=0
MOVL C00837 V=800.0 PL=0
MOVL C00838 V=800.0 PL=0
MOVL C00839 V=800.0 PL=0
MOVL C00840 V=800.0 PL=0
MOVL C00841 V=800.0 PL=0
MOVL C00842 V=800.0 PL=0
MOVL C00843 V=800.0 PL=0
MOVL C00844 V=800.0 PL=0
MOVL C00845 V=800.0 PL=0
MOVL C00846 V=800.0 PL=0
MOVL C00847 V=800.0 PL=0
MOVL C00848 V=800.0 PL=0
MOVL C00849 V=800.0 PL=0
MOVL C00850 V=800.0 PL=0
MOVL C00851 V=800.0 PL=0
MOVL C00852 V=800.0 PL=0
MOVL C00853 V=800.0 PL=0
MOVL C00854 V=800.0 PL=0
MOVL C00855 V=800.0 PL=0
MOVL C00856 V=800.0 PL=0
MOVL C00857 V=800.0 PL=0
MOVL C00858 V=800.0 PL=0
MOVL C00859 V=800.0 PL=0
MOVL C00860 V=800.0 PL=0
MOVL C00861 V=800.0 PL=0
MOVL C00862 V=800.0 PL=0
MOVL C00863 V=800.0 PL=0
MOVL C00864 V=800.0 PL=0
MOVL C00865 V=800.0 PL=0
MOVL C00866 V=800.0 PL=0
MOVL C00867 V=800.0 PL=0
MOVL C00868 V=800.0 PL=0
MOVL C00869 V=800.0 PL=0
MOVL C00870 V=800.0 PL=0
MOVL C00871 V=800.0 PL=0
MOVL C00872 V=800.0 PL=0
MOVL C00873 V=800.0 PL=0
MOVL C00874 V=800.0 PL=0
MOVL C00875 V=800.0 PL=0
MOVL C00876 V=800.0 PL=0
MOVL C00877 V=800.0 PL=0
MOVL C00878 V=800.0 PL=0
MOVL C00879 V=800.0 PL=0
MOVL C00880 V=800.0 PL=0
MOVL C00881 V=800.0 PL=0
MOVL C00882 V=800.0 PL=0
MOVL C00883 V=800.0 PL=0
MOVL C00884 V=800.0 PL=0
MOVL C00885 V=800.0 PL=0
MOVL C00886 V=800.0 PL=0
MOVL C00887 V=800.0 PL=0
MOVL C00888 V=800.0 PL=0
MOVL C00889 V=800.0 PL=0
MOVL C00890 V=800.0 PL=0
MOVL C00891 V=800.0 PL=0
MOVL C00892 V=800.0 PL=0
MOVL C00893 V=800.0 PL=0
MOVL C00894 V=800.0 PL=0
MOVL C00895 V=800.0 PL=0
MOVL C00896 V=800.0 PL=0
MOVL C00897 V=800.0 PL=0
MOVL C00898 V=800.0 PL=0
MOVL C00899 V=800.0 PL=0
MOVL C00900 V=800.0 PL=0
MOVL C00901 V=800.0 PL=0
MOVL C00902 V=800.0 PL=0
MOVL C00903 V=800.0 PL=0
MOVL C00904 V=800.0 PL=0
MOVL C00905 V=800.0 PL=0
MOVL C00906 V=800.0 PL=0
MOVL C00907 V=800.0 PL=0
MOVL C00908 V=800.0 PL=0
MOVL C00909 V=800.0 PL=0
MOVL C00910 V=800.0 PL=0
MOVL C00911 V=800.0 PL=0
MOVL C00912 V=800.0 PL=0
MOVL C00913 V=800.0 PL=0
MOVL C00914 V=800.0 PL=0
MOVL C00915 V=800.0 PL=0
MOVL C00916 V=800.0 PL=0
MOVL C00917 V=800.0 PL=0
MOVL C00918 V=800.0 PL=0
MOVL C00919 V=800.0 PL=0
MOVL C00920 V=800.0 PL=0
MOVL C00921 V=800.0 PL=0
MOVL C00922 V=800.0 PL=0
MOVL C00923 V=800.0 PL=0
MOVL C00924 V=800.0 PL=0
MOVL C00925 V=800.0 PL=0
MOVL C00926 V=800.0 PL=0
MOVL C00927 V=800.0 PL=0
MOVL C00928 V=800.0 PL=0
MOVL C00929 V=800.0 PL=0
MOVL C00930 V=800.0 PL=0
MOVL C00931 V=800.0 PL=0
MOVL C00932 V=800.0 PL=0
MOVL C00933 V=800.0 PL=0
MOVL C00934 V=800.0 PL=0
MOVL C00935 V=800.0 PL=0
MOVL C00936 V=800.0 PL=0
MOVL C00937 V=800.0 PL=0
MOVL C00938 V=800.0 PL=0
MOVL C00939 V=800.0 PL=0
MOVL C00940 V=800.0 PL=0
MOVL C00941 V=800.0 PL=0
MOVL C00942 V=800.0 PL=0
MOVL C00943 V=800.0 PL=0
MOVL C00944 V=800.0 PL=0
MOVL C00945 V=800.0 PL=0
MOVL C00946 V=800.0 PL=0
MOVL C00947 V=800.0 PL=0
MOVL C00948 V=800.0 PL=0
MOVL C00949 V=800.0 PL=0
MOVL C00950 V=800.0 PL=0
MOVL C00951 V=800.0 PL=0
MOVL C00952 V=800.0 PL=0
MOVL C00953 V=800.0 PL=0
MOVL C00954 V=800.0 PL=0
MOVL C00955 V=800.0 PL=0
MOVL C00956 V=800.0 PL=0
MOVL C00957 V=800.0 PL=0
MOVL C00958 V=800.0 PL=0
MOVL C00959 V=800.0 PL=0
MOVL C00960 V=800.0 PL=0
MOVL C00961 V=800.0 PL=0
MOVL C00962 V=800.0 PL=0
MOVL C00963 V=800.0 PL=0
MOVL C00964 V=800.0 PL=0
MOVL C00965 V=800.0 PL=0
MOVL C00966 V=800.0 PL=0
MOVL C00967 V=800.0 PL=0
MOVL C00968 V=800.0 PL=0
MOVL C00969 V=800.0 PL=0
MOVL C00970 V=800.0 PL=0
MOVL C00971 V=800.0 PL=0
MOVL C00972 V=800.0 PL=0
MOVL C00973 V=800.0 PL=0
MOVL C00974 V=800.0 PL=0
MOVL C00975 V=800.0 PL=0
MOVL C00976 V=800.0 PL=0
MOVL C00977 V=800.0 PL=0
MOVL C00978 V=800.0 PL=0
MOVL C00979 V=800.0 PL=0
MOVL C00980 V=800.0 PL=0
MOVL C00981 V=800.0 PL=0
MOVL C00982 V=800.0 PL=0
MOVL C00983 V=800.0 PL=0
MOVL C00984 V=800.0 PL=0
MOVL C00985 V=800.0 PL=0
MOVL C00986 V=800.0 PL=0
MOVL C00987 V=800.0 PL=0
MOVL C00988 V=800.0 PL=0
MOVL C00989 V=800.0 PL=0
MOVL C00990 V=800.0 PL=0
MOVL C00991 V=800.0 PL=0
MOVL C00992 V=800.0 PL=0
MOVL C00993 V=800.0 PL=0
MOVL C00994 V=800.0 PL=0
MOVL C00995 V=800.0 PL=0
MOVL C00996 V=800.0 PL=0
MOVL C00997 V=800.0 PL=0
MOVL C00998 V=800.0 PL=0
MOVL C00999 V=800.0 PL=0
MOVL C01000 V=800.0 PL=0
MOVL C01001 V=800.0 PL=0
MOVL C01002 V=800.0 PL=0
MOVL C01003 V=800.0 PL=0
MOVL C01004 V=800.0 PL=0
MOVL C01005 V=800.0 PL=0
MOVL C01006 V=800.0 PL=0
MOVL C01007 V=800.0 PL=0
MOVL C01008 V=800.0 PL=0
MOVL C01009 V=800.0 PL=0
MOVL C01010 V=800.0 PL=0
MOVL C01011 V=800.0 PL=0
MOVL C01012 V=800.0 PL=0
MOVL C01013 V=800.0 PL=0
MOVL C01014 V=800.0 PL=0
MOVL C01015 V=800.0 PL=0
MOVL C01016 V=800.0 PL=0
MOVL C01017 V=800.0 PL=0
MOVL C01018 V=800.0 PL=0
MOVL C01019 V=800.0 PL=0
MOVL C01020 V=800.0 PL=0
MOVL C01021 V=800.0 PL=0
MOVL C01022 V=800.0 PL=0
MOVL C01023 V=800.0 PL=0
MOVL C01024 V=800.0 PL=0
MOVL C01025 V=800.0 PL=0
MOVL C01026 V=800.0 PL=0
MOVL C01027 V=800.0 PL=0
MOVL C01028 V=800.0 PL=0
MOVL C01029 V=800.0 PL=0
MOVL C01030 V=800.0 PL=0
MOVL C01031 V=800.0 PL=0
MOVL C01032 V=800.0 PL=0
MOVL C01033 V=800.0 PL=0
MOVL C01034 V=800.0 PL=0
MOVL C01035 V=800.0 PL=0
MOVL C01036 V=800.0 PL=0
MOVL C01037 V=800.0 PL=0
MOVL C01038 V=800.0 PL=0
MOVL C01039 V=800.0 PL=0
MOVL C01040 V=800.0 PL=0
MOVL C01041 V=800.0 PL=0
MOVL C01042 V=800.0 PL=0
MOVL C01043 V=800.0 PL=0
MOVL C01044 V=800.0 PL=0
MOVL C01045 V=800.0 PL=0
MOVL C01046 V=800.0 PL=0
MOVL C01047 V=800.0 PL=0
MOVL C01048 V=800.0 PL=0
MOVL C01049 V=800.0 PL=0
MOVL C01050 V=800.0 PL=0
MOVL C01051 V=800.0 PL=0
MOVL C01052 V=800.0 PL=0
MOVL C01053 V=800.0 PL=0
MOVL C01054 V=800.0 PL=0
MOVL C01055 V=800.0 PL=0
MOVL C01056 V=800.0 PL=0
MOVL C01057 V=800.0 PL=0
MOVL C01058 V=800.0 PL=0
MOVL C01059 V=800.0 PL=0
MOVL C01060 V=800.0 PL=0
MOVL C01061 V=800.0 PL=0
MOVL C01062 V=800.0 PL=0
MOVL C01063 V=800.0 PL=0
MOVL C01064 V=800.0 PL=0
MOVL C01065 V=800.0 PL=0
MOVL C01066 V=800.0 PL=0
MOVL C01067 V=800.0 PL=0
MOVL C01068 V=800.0 PL=0
MOVL C01069 V=800.0 PL=0
MOVL C01070 V=800.0 PL=0
MOVL C01071 V=800.0 PL=0
MOVL C01072 V=800.0 PL=0
MOVL C01073 V=800.0 PL=0
MOVL C01074 V=800.0 PL=0
MOVL C01075 V=800.0 PL=0
MOVL C01076 V=800.0 PL=0
MOVL C01077 V=800.0 PL=0
MOVL C01078 V=800.0 PL=0
MOVL C01079 V=800.0 PL=0
MOVL C01080 V=800.0 PL=0
MOVL C01081 V=800.0 PL=0
MOVL C01082 V=800.0 PL=0
MOVL C01083 V=800.0 PL=0
MOVL C01084 V=800.0 PL=0
MOVL C01085 V=800.0 PL=0
MOVL C01086 V=800.0 PL=0
MOVL C01087 V=800.0 PL=0
MOVL C01088 V=800.0 PL=0
MOVL C01089 V=800.0 PL=0
MOVL C01090 V=800.0 PL=0
MOVL C01091 V=800.0 PL=0
MOVL C01092 V=800.0 PL=0
MOVL C01093 V=800.0 PL=0
MOVL C01094 V=800.0 PL=0
MOVL C01095 V=800.0 PL=0
MOVL C01096 V=800.0 PL=0
MOVL C01097 V=800.0 PL=0
MOVL C01098 V=800.0 PL=0
MOVL C01099 V=800.0 PL=0
MOVL C01100 V=800.0 PL=0
MOVL C01101 V=800.0 PL=0
MOVL C01102 V=800.0 PL=0
MOVL C01103 V=800.0 PL=0
MOVL C01104 V=800.0 PL=0
MOVL C01105 V=800.0 PL=0
MOVL C01106 V=800.0 PL=0
MOVL C01107 V=800.0 PL=0
MOVL C01108 V=800.0 PL=0
MOVL C01109 V=800.0 PL=0
MOVL C01110 V=800.0 PL=0
MOVL C01111 V=800.0 PL=0
MOVL C01112 V=800.0 PL=0
MOVL C01113 V=800.0 PL=0
MOVL C01114 V=800.0 PL=0
MOVL C01115 V=800.0 PL=0
MOVL C01116 V=800.0 PL=0
MOVL C01117 V=800.0 PL=0
MOVL C01118 V=800.0 PL=0
MOVL C01119 V=800.0 PL=0
MOVL C01120 V=800.0 PL=0
MOVL C01121 V=800.0 PL=0
MOVL C01122 V=800.0 PL=0
MOVL C01123 V=800.0 PL=0
MOVL C01124 V=800.0 PL=0
MOVL C01125 V=800.0 PL=0
MOVL C01126 V=800.0 PL=0
MOVL C01127 V=800.0 PL=0
MOVL C01128 V=800.0 PL=0
MOVL C01129 V=800.0 PL=0
MOVL C01130 V=800.0 PL=0
MOVL C01131 V=800.0 PL=0
MOVL C01132 V=800.0 PL=0
MOVL C01133 V=800.0 PL=0
MOVL C01134 V=800.0 PL=0
MOVL C01135 V=800.0 PL=0
MOVL C01136 V=800.0 PL=0
MOVL C01137 V=800.0 PL=0
MOVL C01138 V=800.0 PL=0
MOVL C01139 V=800.0 PL=0
MOVL C01140 V=800.0 PL=0
MOVL C01141 V=800.0 PL=0
MOVL C01142 V=800.0 PL=0
MOVL C01143 V=800.0 PL=0
MOVL C01144 V=800.0 PL=0
MOVL C01145 V=800.0 PL=0
MOVL C01146 V=800.0 PL=0
MOVL C01147 V=800.0 PL=0
MOVL C01148 V=800.0 PL=0
MOVL C01149 V=800.0 PL=0
MOVL C01150 V=800.0 PL=0
MOVL C01151 V=800.0 PL=0
MOVL C01152 V=800.0 PL=0
MOVL C01153 V=800.0 PL=0
MOVL C01154 V=800.0 PL=0
MOVL C01155 V=800.0 PL=0
MOVL C01156 V=800.0 PL=0
MOVL C01157 V=800.0 PL=0
MOVL C01158 V=800.0 PL=0
MOVL C01159 V=800.0 PL=0
MOVL C01160 V=800.0 PL=0
MOVL C01161 V=800.0 PL=0
MOVL C01162 V=800.0 PL=0
MOVL C01163 V=800.0 PL=0
MOVL C01164 V=800.0 PL=0
MOVL C01165 V=800.0 PL=0
MOVL C01166 V=800.0 PL=0
MOVL C01167 V=800.0 PL=0
MOVL C01168 V=800.0 PL=0
MOVL C01169 V=800.0 PL=0
MOVL C01170 V=800.0 PL=0
MOVL C01171 V=800.0 PL=0
MOVL C01172 V=800.0 PL=0
MOVL C01173 V=800.0 PL=0
MOVL C01174 V=800.0 PL=0
MOVL C01175 V=800.0 PL=0
MOVL C01176 V=800.0 PL=0
MOVL C01177 V=800.0 PL=0
MOVL C01178 V=800.0 PL=0
MOVL C01179 V=800.0 PL=0
MOVL C01180 V=800.0 PL=0
MOVL C01181 V=800.0 PL=0
MOVL C01182 V=800.0 PL=0
MOVL C01183 V=800.0 PL=0
MOVL C01184 V=800.0 PL=0
MOVL C01185 V=800.0 PL=0
MOVL C01186 V=800.0 PL=0
MOVL C01187 V=800.0 PL=0
MOVL C01188 V=800.0 PL=0
MOVL C01189 V=800.0 PL=0
MOVL C01190 V=800.0 PL=0
MOVL C01191 V=800.0 PL=0
MOVL C01192 V=800.0 PL=0
MOVL C01193 V=800.0 PL=0
MOVL C01194 V=800.0 PL=0
MOVL C01195 V=800.0 PL=0
MOVL C01196 V=800.0 PL=0
MOVL C01197 V=800.0 PL=0
MOVL C01198 V=800.0 PL=0
MOVL C01199 V=800.0 PL=0
MOVL C01200 V=800.0 PL=0
MOVL C01201 V=800.0 PL=0
MOVL C01202 V=800.0 PL=0
MOVL C01203 V=800.0 PL=0
MOVL C01204 V=800.0 PL=0
MOVL C01205 V=800.0 PL=0
MOVL C01206 V=800.0 PL=0
MOVL C01207 V=800.0 PL=0
MOVL C01208 V=800.0 PL=0
MOVL C01209 V=800.0 PL=0
MOVL C01210 V=800.0 PL=0
MOVL C01211 V=800.0 PL=0
MOVL C01212 V=800.0 PL=0
MOVL C01213 V=800.0 PL=0
MOVL C01214 V=800.0 PL=0
MOVL C01215 V=800.0 PL=0
MOVL C01216 V=800.0 PL=0
MOVL C01217 V=800.0 PL=0
MOVL C01218 V=800.0 PL=0
MOVL C01219 V=800.0 PL=0
MOVL C01220 V=800.0 PL=0
MOVL C01221 V=800.0 PL=0
MOVL C01222 V=800.0 PL=0
MOVL C01223 V=800.0 PL=0
MOVL C01224 V=800.0 PL=0
MOVL C01225 V=800.0 PL=0
MOVL C01226 V=800.0 PL=0
MOVL C01227 V=800.0 PL=0
MOVL C01228 V=800.0 PL=0
MOVL C01229 V=800.0 PL=0
MOVL C01230 V=800.0 PL=0
MOVL C01231 V=800.0 PL=0
MOVL C01232 V=800.0 PL=0
MOVL C01233 V=800.0 PL=0
MOVL C01234 V=800.0 PL=0
MOVL C01235 V=800.0 PL=0
MOVL C01236 V=800.0 PL=0
MOVL C01237 V=800.0 PL=0
MOVL C01238 V=800.0 PL=0
MOVL C01239 V=800.0 PL=0
MOVL C01240 V=800.0 PL=0
MOVL C01241 V=800.0 PL=0
MOVL C01242 V=800.0 PL=0
MOVL C01243 V=800.0 PL=0
MOVL C01244 V=800.0 PL=0
MOVL C01245 V=800.0 PL=0
MOVL C01246 V=800.0 PL=0
MOVL C01247 V=800.0 PL=0
MOVL C01248 V=800.0 PL=0
MOVL C01249 V=800.0 PL=0
MOVL C01250 V=800.0 PL=0
MOVL C01251 V=800.0 PL=0
MOVL C01252 V=800.0 PL=0
MOVL C01253 V=800.0 PL=0
MOVL C01254 V=800.0 PL=0
MOVL C01255 V=800.0 PL=0
MOVL C01256 V=800.0 PL=0
MOVL C01257 V=800.0 PL=0
MOVL C01258 V=800.0 PL=0
MOVL C01259 V=800.0 PL=0
MOVL C01260 V=800.0 PL=0
MOVL C01261 V=800.0 PL=0
MOVL C01262 V=800.0 PL=0
MOVL C01263 V=800.0 PL=0
MOVL C01264 V=800.0 PL=0
MOVL C01265 V=800.0 PL=0
MOVL C01266 V=800.0 PL=0
MOVL C01267 V=800.0 PL=0
MOVL C01268 V=800.0 PL=0
MOVL C01269 V=800.0 PL=0
MOVL C01270 V=800.0 PL=0
MOVL C01271 V=800.0 PL=0
MOVL C01272 V=800.0 PL=0
MOVL C01273 V=800.0 PL=0
MOVL C01274 V=800.0 PL=0
MOVL C01275 V=800.0 PL=0
MOVL C01276 V=800.0 PL=0
MOVL C01277 V=800.0 PL=0
MOVL C01278 V=800.0 PL=0
MOVL C01279 V=800.0 PL=0
MOVL C01280 V=800.0 PL=0
MOVL C01281 V=800.0 PL=0
MOVL C01282 V=800.0 PL=0
MOVL C01283 V=800.0 PL=0
MOVL C01284 V=800.0 PL=0
MOVL C01285 V=800.0 PL=0
MOVL C01286 V=800.0 PL=0
MOVL C01287 V=800.0 PL=0
MOVL C01288 V=800.0 PL=0
MOVL C01289 V=800.0 PL=0
MOVL C01290 V=800.0 PL=0
MOVL C01291 V=800.0 PL=0
MOVL C01292 V=800.0 PL=0
MOVL C01293 V=800.0 PL=0
MOVL C01294 V=800.0 PL=0
MOVL C01295 V=800.0 PL=0
MOVL C01296 V=800.0 PL=0
MOVL C01297 V=800.0 PL=0
MOVL C01298 V=800.0 PL=0
MOVL C01299 V=800.0 PL=0
MOVL C01300 V=800.0 PL=0
MOVL C01301 V=800.0 PL=0
MOVL C01302 V=800.0 PL=0
MOVL C01303 V=800.0 PL=0
MOVL C01304 V=800.0 PL=0
MOVL C01305 V=800.0 PL=0
MOVL C01306 V=800.0 PL=0
MOVL C01307 V=800.0 PL=0
MOVL C01308 V=800.0 PL=0
MOVL C01309 V=800.0 PL=0
MOVL C01310 V=800.0 PL=0
MOVL C01311 V=800.0 PL=0
MOVL C01312 V=800.0 PL=0
MOVL C01313 V=800.0 PL=0
MOVL C01314 V=800.0 PL=0
MOVL C01315 V=800.0 PL=0
MOVL C01316 V=800.0 PL=0
MOVL C01317 V=800.0 PL=0
MOVL C01318 V=800.0 PL=0
MOVL C01319 V=800.0 PL=0
MOVL C01320 V=800.0 PL=0
MOVL C01321 V=800.0 PL=0
MOVL C01322 V=800.0 PL=0
MOVL C01323 V=800.0 PL=0
MOVL C01324 V=800.0 PL=0
MOVL C01325 V=800.0 PL=0
MOVL C01326 V=800.0 PL=0
MOVL C01327 V=800.0 PL=0
MOVL C01328 V=800.0 PL=0
MOVL C01329 V=800.0 PL=0
MOVL C01330 V=800.0 PL=0
MOVL C01331 V=800.0 PL=0
MOVL C01332 V=800.0 PL=0
MOVL C01333 V=800.0 PL=0
MOVL C01334 V=800.0 PL=0
MOVL C01335 V=800.0 PL=0
MOVL C01336 V=800.0 PL=0
MOVL C01337 V=800.0 PL=0
MOVL C01338 V=800.0 PL=0
MOVL C01339 V=800.0 PL=0
MOVL C01340 V=800.0 PL=0
MOVL C01341 V=800.0 PL=0
MOVL C01342 V=800.0 PL=0
MOVL C01343 V=800.0 PL=0
MOVL C01344 V=800.0 PL=0
MOVL C01345 V=800.0 PL=0
MOVL C01346 V=800.0 PL=0
MOVL C01347 V=800.0 PL=0
MOVL C01348 V=800.0 PL=0
MOVL C01349 V=800.0 PL=0
MOVL C01350 V=800.0 PL=0
MOVL C01351 V=800.0 PL=0
MOVL C01352 V=800.0 PL=0
MOVL C01353 V=800.0 PL=0
MOVL C01354 V=800.0 PL=0
MOVL C01355 V=800.0 PL=0
MOVL C01356 V=800.0 PL=0
MOVL C01357 V=800.0 PL=0
MOVL C01358 V=800.0 PL=0
MOVL C01359 V=800.0 PL=0
MOVL C01360 V=800.0 PL=0
MOVL C01361 V=800.0 PL=0
MOVL C01362 V=800.0 PL=0
MOVL C01363 V=800.0 PL=0
MOVL C01364 V=800.0 PL=0
MOVL C01365 V=800.0 PL=0
MOVL C01366 V=800.0 PL=0
MOVL C01367 V=800.0 PL=0
MOVL C01368 V=800.0 PL=0
MOVL C01369 V=800.0 PL=0
MOVL C01370 V=800.0 PL=0
MOVL C01371 V=800.0 PL=0
MOVL C01372 V=800.0 PL=0
MOVL C01373 V=800.0 PL=0
MOVL C01374 V=800.0 PL=0
MOVL C01375 V=800.0 PL=0
MOVL C01376 V=800.0 PL=0
MOVL C01377 V=800.0 PL=0
MOVL C01378 V=800.0 PL=0
MOVL C01379 V=800.0 PL=0
MOVL C01380 V=800.0 PL=0
MOVL C01381 V=800.0 PL=0
MOVL C01382 V=800.0 PL=0
MOVL C01383 V=800.0 PL=0
MOVL C01384 V=800.0 PL=0
MOVL C01385 V=800.0 PL=0
MOVL C01386 V=800.0 PL=0
MOVL C01387 V=800.0 PL=0
MOVL C01388 V=800.0 PL=0
MOVL C01389 V=800.0 PL=0
MOVL C01390 V=800.0 PL=0
MOVL C01391 V=800.0 PL=0
MOVL C01392 V=800.0 PL=0
MOVL C01393 V=800.0 PL=0
MOVL C01394 V=800.0 PL=0
MOVL C01395 V=800.0 PL=0
MOVL C01396 V=800.0 PL=0
MOVL C01397 V=800.0 PL=0
MOVL C01398 V=800.0 PL=0
MOVL C01399 V=800.0 PL=0
MOVL C01400 V=800.0 PL=0
MOVL C01401 V=800.0 PL=0
MOVL C01402 V=800.0 PL=0
MOVL C01403 V=800.0 PL=0
MOVL C01404 V=800.0 PL=0
MOVL C01405 V=800.0 PL=0
MOVL C01406 V=800.0 PL=0
MOVL C01407 V=800.0 PL=0
MOVL C01408 V=800.0 PL=0
MOVL C01409 V=800.0 PL=0
MOVL C01410 V=800.0 PL=0
MOVL C01411 V=800.0 PL=0
MOVL C01412 V=800.0 PL=0
MOVL C01413 V=800.0 PL=0
MOVL C01414 V=800.0 PL=0
MOVL C01415 V=800.0 PL=0
MOVL C01416 V=800.0 PL=0
MOVL C01417 V=800.0 PL=0
MOVL C01418 V=800.0 PL=0
MOVL C01419 V=800.0 PL=0
MOVL C01420 V=800.0 PL=0
MOVL C01421 V=800.0 PL=0
MOVL C01422 V=800.0 PL=0
MOVL C01423 V=800.0 PL=0
MOVL C01424 V=800.0 PL=0
MOVL C01425 V=800.0 PL=0
MOVL C01426 V=800.0 PL=0
MOVL C01427 V=800.0 PL=0
MOVL C01428 V=800.0 PL=0
MOVL C01429 V=800.0 PL=0
MOVL C01430 V=800.0 PL=0
MOVL C01431 V=800.0 PL=0
MOVL C01432 V=800.0 PL=0
MOVL C01433 V=800.0 PL=0
MOVL C01434 V=800.0 PL=0
MOVL C01435 V=800.0 PL=0
MOVL C01436 V=800.0 PL=0
MOVL C01437 V=800.0 PL=0
MOVL C01438 V=800.0 PL=0
MOVL C01439 V=800.0 PL=0
MOVL C01440 V=800.0 PL=0
MOVL C01441 V=800.0 PL=0
MOVL C01442 V=800.0 PL=0
MOVL C01443 V=800.0 PL=0
MOVL C01444 V=800.0 PL=0
MOVL C01445 V=800.0 PL=0
MOVL C01446 V=800.0 PL=0
MOVL C01447 V=800.0 PL=0
MOVL C01448 V=800.0 PL=0
MOVL C01449 V=800.0 PL=0
MOVL C01450 V=800.0 PL=0
MOVL C01451 V=800.0 PL=0
MOVL C01452 V=800.0 PL=0
MOVL C01453 V=800.0 PL=0
MOVL C01454 V=800.0 PL=0
MOVL C01455 V=800.0 PL=0
MOVL C01456 V=800.0 PL=0
MOVL C01457 V=800.0 PL=0
MOVL C01458 V=800.0 PL=0
MOVL C01459 V=800.0 PL=0
MOVL C01460 V=800.0 PL=0
MOVL C01461 V=800.0 PL=0
MOVL C01462 V=800.0 PL=0
MOVL C01463 V=800.0 PL=0
MOVL C01464 V=800.0 PL=0
MOVL C01465 V=800.0 PL=0
MOVL C01466 V=800.0 PL=0
MOVL C01467 V=800.0 PL=0
MOVL C01468 V=800.0 PL=0
MOVL C01469 V=800.0 PL=0
MOVL C01470 V=800.0 PL=0
MOVL C01471 V=800.0 PL=0
MOVL C01472 V=800.0 PL=0
MOVL C01473 V=800.0 PL=0
MOVL C01474 V=800.0 PL=0
MOVL C01475 V=800.0 PL=0
MOVL C01476 V=800.0 PL=0
MOVL C01477 V=800.0 PL=0
MOVL C01478 V=800.0 PL=0
MOVL C01479 V=800.0 PL=0
MOVL C01480 V=800.0 PL=0
MOVL C01481 V=800.0 PL=0
MOVL C01482 V=800.0 PL=0
MOVL C01483 V=800.0 PL=0
MOVL C01484 V=800.0 PL=0
MOVL C01485 V=800.0 PL=0
MOVL C01486 V=800.0 PL=0
MOVL C01487 V=800.0 PL=0
MOVL C01488 V=800.0 PL=0
MOVL C01489 V=800.0 PL=0
MOVL C01490 V=800.0 PL=0
MOVL C01491 V=800.0 PL=0
MOVL C01492 V=800.0 PL=0
MOVL C01493 V=800.0 PL=0
MOVL C01494 V=800.0 PL=0
MOVL C01495 V=800.0 PL=0
MOVL C01496 V=800.0 PL=0
MOVL C01497 V=800.0 PL=0
MOVL C01498 V=800.0 PL=0
MOVL C01499 V=800.0 PL=0
MOVL C01500 V=800.0 PL=0
MOVL C01501 V=800.0 PL=0
MOVL C01502 V=800.0 PL=0
MOVL C01503 V=800.0 PL=0
MOVL C01504 V=800.0 PL=0
MOVL C01505 V=800.0 PL=0
MOVL C01506 V=800.0 PL=0
MOVL C01507 V=800.0 PL=0
MOVL C01508 V=800.0 PL=0
MOVL C01509 V=800.0 PL=0
MOVL C01510 V=800.0 PL=0
MOVL C01511 V=800.0 PL=0
MOVL C01512 V=800.0 PL=0
MOVL C01513 V=800.0 PL=0
MOVL C01514 V=800.0 PL=0
MOVL C01515 V=800.0 PL=0
MOVL C01516 V=800.0 PL=0
MOVL C01517 V=800.0 PL=0
MOVL C01518 V=800.0 PL=0
MOVL C01519 V=800.0 PL=0
MOVL C01520 V=800.0 PL=0
MOVL C01521 V=800.0 PL=0
MOVL C01522 V=800.0 PL=0
MOVL C01523 V=800.0 PL=0
MOVL C01524 V=800.0 PL=0
MOVL C01525 V=800.0 PL=0
MOVL C01526 V=800.0 PL=0
MOVL C01527 V=800.0 PL=0
MOVL C01528 V=800.0 PL=0
MOVL C01529 V=800.0 PL=0
MOVL C01530 V=800.0 PL=0
MOVL C01531 V=800.0 PL=0
MOVL C01532 V=800.0 PL=0
MOVL C01533 V=800.0 PL=0
MOVL C01534 V=800.0 PL=0
MOVL C01535 V=800.0 PL=0
MOVL C01536 V=800.0 PL=0
MOVL C01537 V=800.0 PL=0
MOVL C01538 V=800.0 PL=0
MOVL C01539 V=800.0 PL=0
MOVL C01540 V=800.0 PL=0
MOVL C01541 V=800.0 PL=0
MOVL C01542 V=800.0 PL=0
MOVL C01543 V=800.0 PL=0
MOVL C01544 V=800.0 PL=0
MOVL C01545 V=800.0 PL=0
MOVL C01546 V=800.0 PL=0
MOVL C01547 V=800.0 PL=0
MOVL C01548 V=800.0 PL=0
MOVL C01549 V=800.0 PL=0
MOVL C01550 V=800.0 PL=0
MOVL C01551 V=800.0 PL=0
MOVL C01552 V=800.0 PL=0
MOVL C01553 V=800.0 PL=0
MOVL C01554 V=800.0 PL=0
MOVL C01555 V=800.0 PL=0
MOVL C01556 V=800.0 PL=0
MOVL C01557 V=800.0 PL=0
MOVL C01558 V=800.0 PL=0
MOVL C01559 V=800.0 PL=0
MOVL C01560 V=800.0 PL=0
MOVL C01561 V=800.0 PL=0
MOVL C01562 V=800.0 PL=0
MOVL C01563 V=800.0 PL=0
MOVL C01564 V=800.0 PL=0
MOVL C01565 V=800.0 PL=0
MOVL C01566 V=800.0 PL=0
MOVL C01567 V=800.0 PL=0
MOVL C01568 V=800.0 PL=0
MOVL C01569 V=800.0 PL=0
MOVL C01570 V=800.0 PL=0
MOVL C01571 V=800.0 PL=0
MOVL C01572 V=800.0 PL=0
MOVL C01573 V=800.0 PL=0
MOVL C01574 V=800.0 PL=0
MOVL C01575 V=800.0 PL=0
MOVL C01576 V=800.0 PL=0
MOVL C01577 V=800.0 PL=0
MOVL C01578 V=800.0 PL=0
MOVL C01579 V=800.0 PL=0
MOVL C01580 V=800.0 PL=0
MOVL C01581 V=800.0 PL=0
MOVL C01582 V=800.0 PL=0
MOVL C01583 V=800.0 PL=0
MOVL C01584 V=800.0 PL=0
MOVL C01585 V=800.0 PL=0
MOVL C01586 V=800.0 PL=0
MOVL C01587 V=800.0 PL=0
MOVL C01588 V=800.0 PL=0
MOVL C01589 V=800.0 PL=0
MOVL C01590 V=800.0 PL=0
MOVL C01591 V=800.0 PL=0
MOVL C01592 V=800.0 PL=0
MOVL C01593 V=800.0 PL=0
MOVL C01594 V=800.0 PL=0
MOVL C01595 V=800.0 PL=0
MOVL C01596 V=800.0 PL=0
MOVL C01597 V=800.0 PL=0
MOVL C01598 V=800.0 PL=0
MOVL C01599 V=800.0 PL=0
MOVL C01600 V=800.0 PL=0
MOVL C01601 V=800.0 PL=0
MOVL C01602 V=800.0 PL=0
MOVL C01603 V=800.0 PL=0
MOVL C01604 V=800.0 PL=0
MOVL C01605 V=800.0 PL=0
MOVL C01606 V=800.0 PL=0
MOVL C01607 V=800.0 PL=0
MOVL C01608 V=800.0 PL=0
MOVL C01609 V=800.0 PL=0
MOVL C01610 V=800.0 PL=0
MOVL C01611 V=800.0 PL=0
MOVL C01612 V=800.0 PL=0
MOVL C01613 V=800.0 PL=0
MOVL C01614 V=800.0 PL=0
MOVL C01615 V=800.0 PL=0
MOVL C01616 V=800.0 PL=0
MOVL C01617 V=800.0 PL=0
MOVL C01618 V=800.0 PL=0
MOVL C01619 V=800.0 PL=0
MOVL C01620 V=800.0 PL=0
MOVL C01621 V=800.0 PL=0
MOVL C01622 V=800.0 PL=0
MOVL C01623 V=800.0 PL=0
MOVL C01624 V=800.0 PL=0
MOVL C01625 V=800.0 PL=0
MOVL C01626 V=800.0 PL=0
MOVL C01627 V=800.0 PL=0
MOVL C01628 V=800.0 PL=0
MOVL C01629 V=800.0 PL=0
MOVL C01630 V=800.0 PL=0
MOVL C01631 V=800.0 PL=0
MOVL C01632 V=800.0 PL=0
MOVL C01633 V=800.0 PL=0
MOVL C01634 V=800.0 PL=0
MOVL C01635 V=800.0 PL=0
MOVL C01636 V=800.0 PL=0
MOVL C01637 V=800.0 PL=0
MOVL C01638 V=800.0 PL=0
MOVL C01639 V=800.0 PL=0
MOVL C01640 V=800.0 PL=0
MOVL C01641 V=800.0 PL=0
MOVL C01642 V=800.0 PL=0
MOVL C01643 V=800.0 PL=0
MOVL C01644 V=800.0 PL=0
MOVL C01645 V=800.0 PL=0
MOVL C01646 V=800.0 PL=0
MOVL C01647 V=800.0 PL=0
MOVL C01648 V=800.0 PL=0
MOVL C01649 V=800.0 PL=0
MOVL C01650 V=800.0 PL=0
MOVL C01651 V=800.0 PL=0
MOVL C01652 V=800.0 PL=0
MOVL C01653 V=800.0 PL=0
MOVL C01654 V=800.0 PL=0
MOVL C01655 V=800.0 PL=0
MOVL C01656 V=800.0 PL=0
MOVL C01657 V=800.0 PL=0
MOVL C01658 V=800.0 PL=0
MOVL C01659 V=800.0 PL=0
MOVL C01660 V=800.0 PL=0
MOVL C01661 V=800.0 PL=0
MOVL C01662 V=800.0 PL=0
MOVL C01663 V=800.0 PL=0
MOVL C01664 V=800.0 PL=0
MOVL C01665 V=800.0 PL=0
MOVL C01666 V=800.0 PL=0
MOVL C01667 V=800.0 PL=0
MOVL C01668 V=800.0 PL=0
MOVL C01669 V=800.0 PL=0
MOVL C01670 V=800.0 PL=0
MOVL C01671 V=800.0 PL=0
MOVL C01672 V=800.0 PL=0
MOVL C01673 V=800.0 PL=0
MOVL C01674 V=800.0 PL=0
MOVL C01675 V=800.0 PL=0
MOVL C01676 V=800.0 PL=0
MOVL C01677 V=800.0 PL=0
MOVL C01678 V=800.0 PL=0
MOVL C01679 V=800.0 PL=0
MOVL C01680 V=800.0 PL=0
MOVL C01681 V=800.0 PL=0
MOVL C01682 V=800.0 PL=0
MOVL C01683 V=800.0 PL=0
MOVL C01684 V=800.0 PL=0
MOVL C01685 V=800.0 PL=0
MOVL C01686 V=800.0 PL=0
MOVL C01687 V=800.0 PL=0
MOVL C01688 V=800.0 PL=0
MOVL C01689 V=800.0 PL=0
MOVL C01690 V=800.0 PL=0
MOVL C01691 V=800.0 PL=0
MOVL C01692 V=800.0 PL=0
MOVL C01693 V=800.0 PL=0
MOVL C01694 V=800.0 PL=0
MOVL C01695 V=800.0 PL=0
MOVL C01696 V=800.0 PL=0
MOVL C01697 V=800.0 PL=0
MOVL C01698 V=800.0 PL=0
MOVL C01699 V=800.0 PL=0
MOVL C01700 V=800.0 PL=0
MOVL C01701 V=800.0 PL=0
MOVL C01702 V=800.0 PL=0
MOVL C01703 V=800.0 PL=0
MOVL C01704 V=800.0 PL=0
MOVL C01705 V=800.0 PL=0
MOVL C01706 V=800.0 PL=0
MOVL C01707 V=800.0 PL=0
MOVL C01708 V=800.0 PL=0
MOVL C01709 V=800.0 PL=0
MOVL C01710 V=800.0 PL=0
MOVL C01711 V=800.0 PL=0
MOVL C01712 V=800.0 PL=0
MOVL C01713 V=800.0 PL=0
MOVL C01714 V=800.0 PL=0
MOVL C01715 V=800.0 PL=0
MOVL C01716 V=800.0 PL=0
MOVL C01717 V=800.0 PL=0
MOVL C01718 V=800.0 PL=0
MOVL C01719 V=800.0 PL=0
MOVL C01720 V=800.0 PL=0
MOVL C01721 V=800.0 PL=0
MOVL C01722 V=800.0 PL=0
MOVL C01723 V=800.0 PL=0
MOVL C01724 V=800.0 PL=0
MOVL C01725 V=800.0 PL=0
MOVL C01726 V=800.0 PL=0
MOVL C01727 V=800.0 PL=0
MOVL C01728 V=800.0 PL=0
MOVL C01729 V=800.0 PL=0
MOVL C01730 V=800.0 PL=0
MOVL C01731 V=800.0 PL=0
MOVL C01732 V=800.0 PL=0
MOVL C01733 V=800.0 PL=0
MOVL C01734 V=800.0 PL=0
MOVL C01735 V=800.0 PL=0
MOVL C01736 V=800.0 PL=0
MOVL C01737 V=800.0 PL=0
MOVL C01738 V=800.0 PL=0
MOVL C01739 V=800.0 PL=0
MOVL C01740 V=800.0 PL=0
MOVL C01741 V=800.0 PL=0
MOVL C01742 V=800.0 PL=0
MOVL C01743 V=800.0 PL=0
MOVL C01744 V=800.0 PL=0
MOVL C01745 V=800.0 PL=0
MOVL C01746 V=800.0 PL=0
MOVL C01747 V=800.0 PL=0
MOVL C01748 V=800.0 PL=0
MOVL C01749 V=800.0 PL=0
MOVL C01750 V=800.0 PL=0
MOVL C01751 V=800.0 PL=0
MOVL C01752 V=800.0 PL=0
MOVL C01753 V=800.0 PL=0
MOVL C01754 V=800.0 PL=0
MOVL C01755 V=800.0 PL=0
MOVL C01756 V=800.0 PL=0
MOVL C01757 V=800.0 PL=0
MOVL C01758 V=800.0 PL=0
MOVL C01759 V=800.0 PL=0
MOVL C01760 V=800.0 PL=0
MOVL C01761 V=800.0 PL=0
MOVL C01762 V=800.0 PL=0
MOVL C01763 V=800.0 PL=0
MOVL C01764 V=800.0 PL=0
MOVL C01765 V=800.0 PL=0
MOVL C01766 V=800.0 PL=0
MOVL C01767 V=800.0 PL=0
MOVL C01768 V=800.0 PL=0
MOVL C01769 V=800.0 PL=0
MOVL C01770 V=800.0 PL=0
MOVL C01771 V=800.0 PL=0
MOVL C01772 V=800.0 PL=0
MOVL C01773 V=800.0 PL=0
MOVL C01774 V=800.0 PL=0
MOVL C01775 V=800.0 PL=0
MOVL C01776 V=800.0 PL=0
MOVL C01777 V=800.0 PL=0
MOVL C01778 V=800.0 PL=0
MOVL C01779 V=800.0 PL=0
MOVL C01780 V=800.0 PL=0
MOVL C01781 V=800.0 PL=0
MOVL C01782 V=800.0 PL=0
MOVL C01783 V=800.0 PL=0
MOVL C01784 V=800.0 PL=0
MOVL C01785 V=800.0 PL=0
MOVL C01786 V=800.0 PL=0
MOVL C01787 V=800.0 PL=0
MOVL C01788 V=800.0 PL=0
MOVL C01789 V=800.0 PL=0
MOVL C01790 V=800.0 PL=0
MOVL C01791 V=800.0 PL=0
MOVL C01792 V=800.0 PL=0
MOVL C01793 V=800.0 PL=0
MOVL C01794 V=800.0 PL=0
MOVL C01795 V=800.0 PL=0
MOVL C01796 V=800.0 PL=0
MOVL C01797 V=800.0 PL=0
MOVL C01798 V=800.0 PL=0
MOVL C01799 V=800.0 PL=0
MOVL C01800 V=800.0 PL=0
MOVL C01801 V=800.0 PL=0
MOVL C01802 V=800.0 PL=0
MOVL C01803 V=800.0 PL=0
MOVL C01804 V=800.0 PL=0
MOVL C01805 V=800.0 PL=0
MOVL C01806 V=800.0 PL=0
MOVL C01807 V=800.0 PL=0
MOVL C01808 V=800.0 PL=0
MOVL C01809 V=800.0 PL=0
MOVL C01810 V=800.0 PL=0
MOVL C01811 V=800.0 PL=0
MOVL C01812 V=800.0 PL=0
MOVL C01813 V=800.0 PL=0
MOVL C01814 V=800.0 PL=0
MOVL C01815 V=800.0 PL=0
MOVL C01816 V=800.0 PL=0
MOVL C01817 V=800.0 PL=0
MOVL C01818 V=800.0 PL=0
MOVL C01819 V=800.0 PL=0
MOVL C01820 V=800.0 PL=0
MOVL C01821 V=800.0 PL=0
MOVL C01822 V=800.0 PL=0
MOVL C01823 V=800.0 PL=0
MOVL C01824 V=800.0 PL=0
MOVL C01825 V=800.0 PL=0
MOVL C01826 V=800.0 PL=0
MOVL C01827 V=800.0 PL=0
MOVL C01828 V=800.0 PL=0
MOVL C01829 V=800.0 PL=0
MOVL C01830 V=800.0 PL=0
MOVL C01831 V=800.0 PL=0
MOVL C01832 V=800.0 PL=0
MOVL C01833 V=800.0 PL=0
MOVL C01834 V=800.0 PL=0
MOVL C01835 V=800.0 PL=0
MOVL C01836 V=800.0 PL=0
MOVL C01837 V=800.0 PL=0
MOVL C01838 V=800.0 PL=0
MOVL C01839 V=800.0 PL=0
MOVL C01840 V=800.0 PL=0
MOVL C01841 V=800.0 PL=0
MOVL C01842 V=800.0 PL=0
MOVL C01843 V=800.0 PL=0
MOVL C01844 V=800.0 PL=0
MOVL C01845 V=800.0 PL=0
MOVL C01846 V=800.0 PL=0
MOVL C01847 V=800.0 PL=0
MOVL C01848 V=800.0 PL=0
MOVL C01849 V=800.0 PL=0
MOVL C01850 V=800.0 PL=0
MOVL C01851 V=800.0 PL=0
MOVL C01852 V=800.0 PL=0
MOVL C01853 V=800.0 PL=0
MOVL C01854 V=800.0 PL=0
MOVL C01855 V=800.0 PL=0
MOVL C01856 V=800.0 PL=0
MOVL C01857 V=800.0 PL=0
MOVL C01858 V=800.0 PL=0
MOVL C01859 V=800.0 PL=0
MOVL C01860 V=800.0 PL=0
MOVL C01861 V=800.0 PL=0
MOVL C01862 V=800.0 PL=0
MOVL C01863 V=800.0 PL=0
MOVL C01864 V=800.0 PL=0
MOVL C01865 V=800.0 PL=0
MOVL C01866 V=800.0 PL=0
MOVL C01867 V=800.0 PL=0
MOVL C01868 V=800.0 PL=0
MOVL C01869 V=800.0 PL=0
MOVL C01870 V=800.0 PL=0
MOVL C01871 V=800.0 PL=0
MOVL C01872 V=800.0 PL=0
MOVL C01873 V=800.0 PL=0
MOVL C01874 V=800.0 PL=0
MOVL C01875 V=800.0 PL=0
MOVL C01876 V=800.0 PL=0
MOVL C01877 V=800.0 PL=0
MOVL C01878 V=800.0 PL=0
MOVL C01879 V=800.0 PL=0
MOVL C01880 V=800.0 PL=0
MOVL C01881 V=800.0 PL=0
MOVL C01882 V=800.0 PL=0
MOVL C01883 V=800.0 PL=0
MOVL C01884 V=800.0 PL=0
MOVL C01885 V=800.0 PL=0
MOVL C01886 V=800.0 PL=0
MOVL C01887 V=800.0 PL=0
MOVL C01888 V=800.0 PL=0
MOVL C01889 V=800.0 PL=0
MOVL C01890 V=800.0 PL=0
MOVL C01891 V=800.0 PL=0
MOVL C01892 V=800.0 PL=0
MOVL C01893 V=800.0 PL=0
MOVL C01894 V=800.0 PL=0
MOVL C01895 V=800.0 PL=0
MOVL C01896 V=800.0 PL=0
MOVL C01897 V=800.0 PL=0
MOVL C01898 V=800.0 PL=0
MOVL C01899 V=800.0 PL=0
MOVL C01900 V=800.0 PL=0
MOVL C01901 V=800.0 PL=0
MOVL C01902 V=800.0 PL=0
MOVL C01903 V=800.0 PL=0
MOVL C01904 V=800.0 PL=0
MOVL C01905 V=800.0 PL=0
MOVL C01906 V=800.0 PL=0
MOVL C01907 V=800.0 PL=0
MOVL C01908 V=800.0 PL=0
MOVL C01909 V=800.0 PL=0
MOVL C01910 V=800.0 PL=0
MOVL C01911 V=800.0 PL=0
MOVL C01912 V=800.0 PL=0
MOVL C01913 V=800.0 PL=0
MOVL C01914 V=800.0 PL=0
MOVL C01915 V=800.0 PL=0
MOVL C01916 V=800.0 PL=0
MOVL C01917 V=800.0 PL=0
MOVL C01918 V=800.0 PL=0
MOVL C01919 V=800.0 PL=0
MOVL C01920 V=800.0 PL=0
MOVL C01921 V=800.0 PL=0
MOVL C01922 V=800.0 PL=0
MOVL C01923 V=800.0 PL=0
MOVL C01924 V=800.0 PL=0
MOVL C01925 V=800.0 PL=0
MOVL C01926 V=800.0 PL=0
MOVL C01927 V=800.0 PL=0
MOVL C01928 V=800.0 PL=0
MOVL C01929 V=800.0 PL=0
MOVL C01930 V=800.0 PL=0
MOVL C01931 V=800.0 PL=0
MOVL C01932 V=800.0 PL=0
MOVL C01933 V=800.0 PL=0
MOVL C01934 V=800.0 PL=0
MOVL C01935 V=800.0 PL=0
MOVL C01936 V=800.0 PL=0
MOVL C01937 V=800.0 PL=0
MOVL C01938 V=800.0 PL=0
MOVL C01939 V=800.0 PL=0
MOVL C01940 V=800.0 PL=0
MOVL C01941 V=800.0 PL=0
MOVL C01942 V=800.0 PL=0
MOVL C01943 V=800.0 PL=0
MOVL C01944 V=800.0 PL=0
MOVL C01945 V=800.0 PL=0
MOVL C01946 V=800.0 PL=0
MOVL C01947 V=800.0 PL=0
MOVL C01948 V=800.0 PL=0
MOVL C01949 V=800.0 PL=0
MOVL C01950 V=800.0 PL=0
MOVL C01951 V=800.0 PL=0
MOVL C01952 V=800.0 PL=0
MOVL C01953 V=800.0 PL=0
MOVL C01954 V=800.0 PL=0
MOVL C01955 V=800.0 PL=0
MOVL C01956 V=800.0 PL=0
MOVL C01957 V=800.0 PL=0
MOVL C01958 V=800.0 PL=0
MOVL C01959 V=800.0 PL=0
MOVL C01960 V=800.0 PL=0
MOVL C01961 V=800.0 PL=0
MOVL C01962 V=800.0 PL=0
MOVL C01963 V=800.0 PL=0
MOVL C01964 V=800.0 PL=0
MOVL C01965 V=800.0 PL=0
MOVL C01966 V=800.0 PL=0
MOVL C01967 V=800.0 PL=0
MOVL C01968 V=800.0 PL=0
MOVL C01969 V=800.0 PL=0
MOVL C01970 V=800.0 PL=0
MOVL C01971 V=800.0 PL=0
MOVL C01972 V=800.0 PL=0
MOVL C01973 V=800.0 PL=0
MOVL C01974 V=800.0 PL=0
MOVL C01975 V=800.0 PL=0
MOVL C01976 V=800.0 PL=0
MOVL C01977 V=800.0 PL=0
MOVL C01978 V=800.0 PL=0
MOVL C01979 V=800.0 PL=0
MOVL C01980 V=800.0 PL=0
MOVL C01981 V=800.0 PL=0
MOVL C01982 V=800.0 PL=0
MOVL C01983 V=800.0 PL=0
MOVL C01984 V=800.0 PL=0
MOVL C01985 V=800.0 PL=0
MOVL C01986 V=800.0 PL=0
MOVL C01987 V=800.0 PL=0
MOVL C01988 V=800.0 PL=0
MOVL C01989 V=800.0 PL=0
MOVL C01990 V=800.0 PL=0
MOVL C01991 V=800.0 PL=0
MOVL C01992 V=800.0 PL=0
MOVL C01993 V=800.0 PL=0
MOVL C01994 V=800.0 PL=0
MOVL C01995 V=800.0 PL=0
MOVL C01996 V=800.0 PL=0
MOVL C01997 V=800.0 PL=0
MOVL C01998 V=800.0 PL=0
MOVL C01999 V=800.0 PL=0
MOVL C02000 V=800.0 PL=0
MOVL C02001 V=800.0 PL=0
MOVL C02002 V=800.0 PL=0
MOVL C02003 V=800.0 PL=0
MOVL C02004 V=800.0 PL=0
MOVL C02005 V=800.0 PL=0
MOVL C02006 V=800.0 PL=0
MOVL C02007 V=800.0 PL=0
MOVL C02008 V=800.0 PL=0
MOVL C02009 V=800.0 PL=0
MOVL C02010 V=800.0 PL=0
MOVL C02011 V=800.0 PL=0
MOVL C02012 V=800.0 PL=0
MOVL C02013 V=800.0 PL=0
MOVL C02014 V=800.0 PL=0
MOVL C02015 V=800.0 PL=0
MOVL C02016 V=800.0 PL=0
MOVL C02017 V=800.0 PL=0
MOVL C02018 V=800.0 PL=0
MOVL C02019 V=800.0 PL=0
MOVL C02020 V=800.0 PL=0
MOVL C02021 V=800.0 PL=0
MOVL C02022 V=800.0 PL=0
MOVL C02023 V=800.0 PL=0
MOVL C02024 V=800.0 PL=0
MOVL C02025 V=800.0 PL=0
MOVL C02026 V=800.0 PL=0
MOVL C02027 V=800.0 PL=0
MOVL C02028 V=800.0 PL=0
MOVL C02029 V=800.0 PL=0
MOVL C02030 V=800.0 PL=0
MOVL C02031 V=800.0 PL=0
MOVL C02032 V=800.0 PL=0
MOVL C02033 V=800.0 PL=0
MOVL C02034 V=800.0 PL=0
MOVL C02035 V=800.0 PL=0
MOVL C02036 V=800.0 PL=0
MOVL C02037 V=800.0 PL=0
MOVL C02038 V=800.0 PL=0
MOVL C02039 V=800.0 PL=0
MOVL C02040 V=800.0 PL=0
MOVL C02041 V=800.0 PL=0
MOVL C02042 V=800.0 PL=0
MOVL C02043 V=800.0 PL=0
MOVL C02044 V=800.0 PL=0
MOVL C02045 V=800.0 PL=0
MOVL C02046 V=800.0 PL=0
MOVL C02047 V=800.0 PL=0
MOVL C02048 V=800.0 PL=0
MOVL C02049 V=800.0 PL=0
MOVL C02050 V=800.0 PL=0
MOVL C02051 V=800.0 PL=0
MOVL C02052 V=800.0 PL=0
MOVL C02053 V=800.0 PL=0
MOVL C02054 V=800.0 PL=0
MOVL C02055 V=800.0 PL=0
MOVL C02056 V=800.0 PL=0
MOVL C02057 V=800.0 PL=0
MOVL C02058 V=800.0 PL=0
MOVL C02059 V=800.0 PL=0
MOVL C02060 V=800.0 PL=0
MOVL C02061 V=800.0 PL=0
MOVL C02062 V=800.0 PL=0
MOVL C02063 V=800.0 PL=0
MOVL C02064 V=800.0 PL=0
MOVL C02065 V=800.0 PL=0
MOVL C02066 V=800.0 PL=0
MOVL C02067 V=800.0 PL=0
MOVL C02068 V=800.0 PL=0
MOVL C02069 V=800.0 PL=0
MOVL C02070 V=800.0 PL=0
MOVL C02071 V=800.0 PL=0
MOVL C02072 V=800.0 PL=0
MOVL C02073 V=800.0 PL=0
MOVL C02074 V=800.0 PL=0
MOVL C02075 V=800.0 PL=0
MOVL C02076 V=800.0 PL=0
MOVL C02077 V=800.0 PL=0
MOVL C02078 V=800.0 PL=0
MOVL C02079 V=800.0 PL=0
MOVL C02080 V=800.0 PL=0
MOVL C02081 V=800.0 PL=0
MOVL C02082 V=800.0 PL=0
MOVL C02083 V=800.0 PL=0
MOVL C02084 V=800.0 PL=0
MOVL C02085 V=800.0 PL=0
MOVL C02086 V=800.0 PL=0
MOVL C02087 V=800.0 PL=0
MOVL C02088 V=800.0 PL=0
MOVL C02089 V=800.0 PL=0
MOVL C02090 V=800.0 PL=0
MOVL C02091 V=800.0 PL=0
MOVL C02092 V=800.0 PL=0
MOVL C02093 V=800.0 PL=0
MOVL C02094 V=800.0 PL=0
MOVL C02095 V=800.0 PL=0
MOVL C02096 V=800.0 PL=0
MOVL C02097 V=800.0 PL=0
MOVL C02098 V=800.0 PL=0
MOVL C02099 V=800.0 PL=0
MOVL C02100 V=800.0 PL=0
MOVL C02101 V=800.0 PL=0
MOVL C02102 V=800.0 PL=0
MOVL C02103 V=800.0 PL=0
MOVL C02104 V=800.0 PL=0
MOVL C02105 V=800.0 PL=0
MOVL C02106 V=800.0 PL=0
MOVL C02107 V=800.0 PL=0
MOVL C02108 V=800.0 PL=0
MOVL C02109 V=800.0 PL=0
MOVL C02110 V=800.0 PL=0
MOVL C02111 V=800.0 PL=0
MOVL C02112 V=800.0 PL=0
MOVL C02113 V=800.0 PL=0
MOVL C02114 V=800.0 PL=0
MOVL C02115 V=800.0 PL=0
MOVL C02116 V=800.0 PL=0
MOVL C02117 V=800.0 PL=0
MOVL C02118 V=800.0 PL=0
MOVL C02119 V=800.0 PL=0
MOVL C02120 V=800.0 PL=0
MOVL C02121 V=800.0 PL=0
MOVL C02122 V=800.0 PL=0
MOVL C02123 V=800.0 PL=0
MOVL C02124 V=800.0 PL=0
MOVL C02125 V=800.0 PL=0
MOVL C02126 V=800.0 PL=0
MOVL C02127 V=800.0 PL=0
